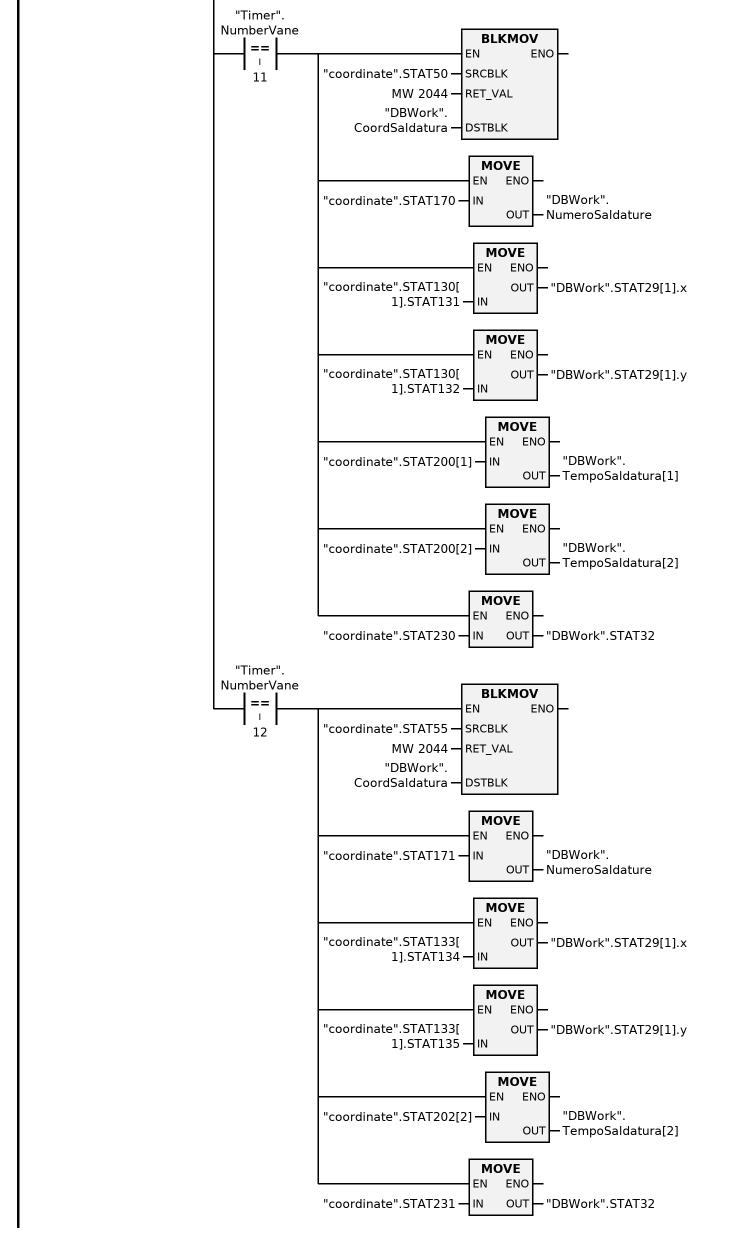
[picture p72: FC51 - TYPE TOOL networks 12-12]
NETWORK
TITLE =
      A     "Type_PP2_9_vane";
      A     "T45";
      =     L 0.0;
      A     L 0.0;
      A(;
      L     "Timer".NumberVane;
      L     9;
      ==I;
      );
      =     L 0.1;
      A     L 0.1;
      JNB   _04f;
      CALL  "BLKMOV" (
           SRCBLK                   := "coordinate".STAT40,
           RET_VAL                  := MW 2044,
           DSTBLK                   := "DBWork".CoordSaldatura);
_04f: NOP   0;
      A     L 0.1;
      JNB   _050;
      L     "coordinate".STAT168;
      T     "DBWork".NumeroSaldature;
_050: NOP   0;
      A     L 0.1;
      JNB   _051;
      L     "coordinate".STAT124[1].STAT125;
      T     "DBWork".STAT29[1].x;
_051: NOP   0;
      A     L 0.1;
      JNB   _052;
      L     "coordinate".STAT124[1].STAT126;
      T     "DBWork".STAT29[1].y;
_052: NOP   0;
      A     L 0.1;
      JNB   _053;
      L     "coordinate".STAT196[1];
      T     "DBWork".TempoSaldatura[1];
_053: NOP   0;
      A     L 0.1;
      JNB   _054;
      L     "coordinate".STAT196[2];
      T     "DBWork".TempoSaldatura[2];
_054: NOP   0;
      A     L 0.1;
      JNB   _055;
      L     "coordinate".STAT228;
      T     "DBWork".STAT32;
_055: NOP   0;
      A     L 0.0;
      A(;
      L     "Timer".NumberVane;
      L     10;
      ==I;
      );
      =     L 0.1;
      A     L 0.1;
      JNB   _056;
      CALL  "BLKMOV" (
           SRCBLK                   := "coordinate".STAT45,
           RET_VAL                  := MW 2044,
           DSTBLK                   := "DBWork".CoordSaldatura);
_056: NOP   0;
      A     L 0.1;
      JNB   _057;
      L     "coordinate".STAT169;
      T     "DBWork".NumeroSaldature;
_057: NOP   0;
      A     L 0.1;
      JNB   _058;
      L     "coordinate".STAT127[1].STAT128;
      T     "DBWork".STAT29[1].x;
_058: NOP   0;
      A     L 0.1;
      JNB   _059;
      L     "coordinate".STAT127[1].STAT129;
      T     "DBWork".STAT29[1].y;
_059: NOP   0;
      A     L 0.1;
      JNB   _05a;
      L     "coordinate".STAT198[1];
      T     "DBWork".TempoSaldatura[1];
_05a: NOP   0;
      A     L 0.1;
      JNB   _05b;
      L     "coordinate".STAT198[2];
      T     "DBWork".TempoSaldatura[2];
_05b: NOP   0;
      A     L 0.1;
      JNB   _05c;
      L     "coordinate".STAT229;
      T     "DBWork".STAT32;
_05c: NOP   0;
      A     L 0.0;
      A(;
      L     "Timer".NumberVane;
      L     11;
      ==I;
      );
      =     L 0.1;
      A     L 0.1;
      JNB   _05d;
      CALL  "BLKMOV" (
           SRCBLK                   := "coordinate".STAT50,
           RET_VAL                  := MW 2044,
           DSTBLK                   := "DBWork".CoordSaldatura);
_05d: NOP   0;
      A     L 0.1;
      JNB   _05e;
      L     "coordinate".STAT170;
      T     "DBWork".NumeroSaldature;
_05e: NOP   0;
      A     L 0.1;
      JNB   _05f;
      L     "coordinate".STAT130[1].STAT131;
      T     "DBWork".STAT29[1].x;
_05f: NOP   0;
      A     L 0.1;
      JNB   _060;
      L     "coordinate".STAT130[1].STAT132;
      T     "DBWork".STAT29[1].y;
_060: NOP   0;
      A     L 0.1;
      JNB   _061;
      L     "coordinate".STAT200[1];
      T     "DBWork".TempoSaldatura[1];
_061: NOP   0;
      A     L 0.1;
      JNB   _062;
      L     "coordinate".STAT200[2];
      T     "DBWork".TempoSaldatura[2];
_062: NOP   0;
      A     L 0.1;
      JNB   _063;
      L     "coordinate".STAT230;
      T     "DBWork".STAT32;
_063: NOP   0;
      A     L 0.0;
      A(;
      L     "Timer".NumberVane;
      L     12;
      ==I;
      );
      =     L 0.1;
      A     L 0.1;
      JNB   _064;
      CALL  "BLKMOV" (
           SRCBLK                   := "coordinate".STAT55,
           RET_VAL                  := MW 2044,
           DSTBLK                   := "DBWork".CoordSaldatura);
_064: NOP   0;
      A     L 0.1;
      JNB   _065;
      L     "coordinate".STAT171;
      T     "DBWork".NumeroSaldature;
_065: NOP   0;
      A     L 0.1;
      JNB   _066;
      L     "coordinate".STAT133[1].STAT134;
      T     "DBWork".STAT29[1].x;
_066: NOP   0;
      A     L 0.1;
      JNB   _067;
      L     "coordinate".STAT133[1].STAT135;
      T     "DBWork".STAT29[1].y;
_067: NOP   0;
      A     L 0.1;
      JNB   _068;
      L     "coordinate".STAT202[2];
      T     "DBWork".TempoSaldatura[2];
_068: NOP   0;
      A     L 0.1;
      JNB   _069;
      L     "coordinate".STAT231;
      T     "DBWork".STAT32;
_069: NOP   0;
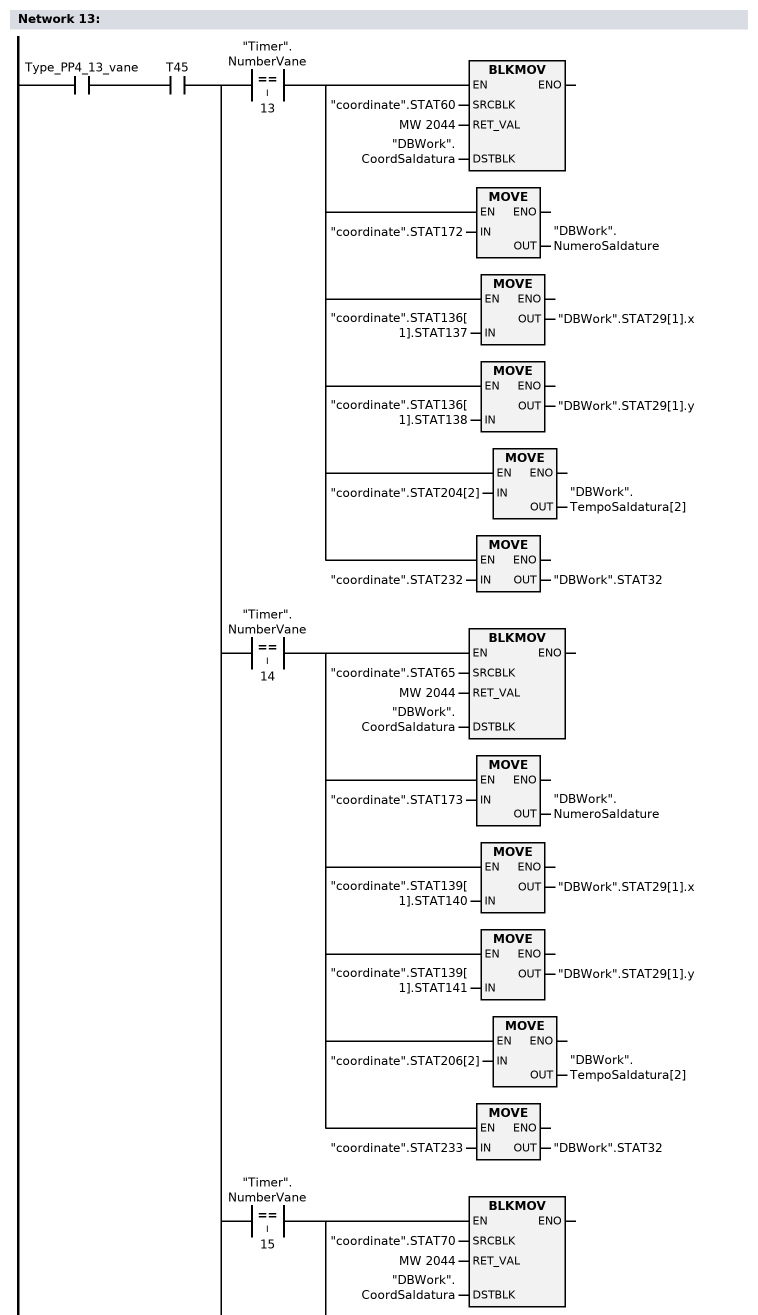
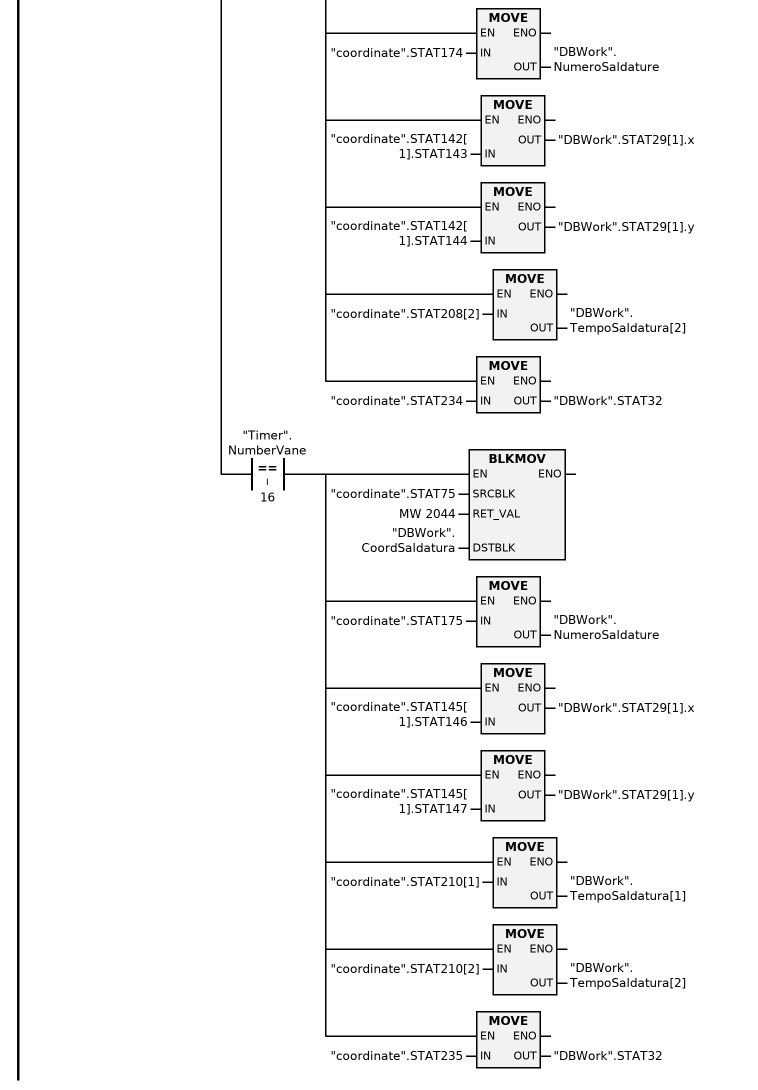
NETWORK
TITLE =
      A     "Type_PP4_13_vane";
      A     "T45";
      =     L 0.0;
      A     L 0.0;
      A(;
      L     "Timer".NumberVane;
      L     13;
      ==I;
      );
      =     L 0.1;
      A     L 0.1;
      JNB   _06a;
      CALL  "BLKMOV" (
           SRCBLK                   := "coordinate".STAT60,
           RET_VAL                  := MW 2044,
           DSTBLK                   := "DBWork".CoordSaldatura);
_06a: NOP   0;
      A     L 0.1;
      JNB   _06b;
      L     "coordinate".STAT172;
      T     "DBWork".NumeroSaldature;
_06b: NOP   0;
      A     L 0.1;
      JNB   _06c;
      L     "coordinate".STAT136[1].STAT137;
      T     "DBWork".STAT29[1].x;
_06c: NOP   0;
      A     L 0.1;
      JNB   _06d;
      L     "coordinate".STAT136[1].STAT138;
      T     "DBWork".STAT29[1].y;
_06d: NOP   0;
      A     L 0.1;
      JNB   _06e;
      L     "coordinate".STAT204[2];
      T     "DBWork".TempoSaldatura[2];
_06e: NOP   0;
      A     L 0.1;
      JNB   _06f;
      L     "coordinate".STAT232;
      T     "DBWork".STAT32;
_06f: NOP   0;
      A     L 0.0;
      A(;
      L     "Timer".NumberVane;
      L     14;
      ==I;
      );
      =     L 0.1;
      A     L 0.1;
      JNB   _070;
      CALL  "BLKMOV" (
           SRCBLK                   := "coordinate".STAT65,
           RET_VAL                  := MW 2044,
           DSTBLK                   := "DBWork".CoordSaldatura);
_070: NOP   0;
      A     L 0.1;
      JNB   _071;
      L     "coordinate".STAT173;
      T     "DBWork".NumeroSaldature;
_071: NOP   0;
      A     L 0.1;
      JNB   _072;
      L     "coordinate".STAT139[1].STAT140;
      T     "DBWork".STAT29[1].x;
_072: NOP   0;
      A     L 0.1;
      JNB   _073;
      L     "coordinate".STAT139[1].STAT141;
      T     "DBWork".STAT29[1].y;
_073: NOP   0;
      A     L 0.1;
      JNB   _074;
      L     "coordinate".STAT206[2];
      T     "DBWork".TempoSaldatura[2];
_074: NOP   0;
      A     L 0.1;
      JNB   _075;
      L     "coordinate".STAT233;
      T     "DBWork".STAT32;
_075: NOP   0;
      A     L 0.0;
      A(;
      L     "Timer".NumberVane;
      L     15;
      ==I;
      );
      =     L 0.1;
      A     L 0.1;
      JNB   _076;
      CALL  "BLKMOV" (
           SRCBLK                   := "coordinate".STAT70,
           RET_VAL                  := MW 2044,
           DSTBLK                   := "DBWork".CoordSaldatura);
_076: NOP   0;
      A     L 0.1;
      JNB   _077;
      L     "coordinate".STAT174;
      T     "DBWork".NumeroSaldature;
_077: NOP   0;
      A     L 0.1;
      JNB   _078;
      L     "coordinate".STAT142[1].STAT143;
      T     "DBWork".STAT29[1].x;
_078: NOP   0;
      A     L 0.1;
      JNB   _079;
      L     "coordinate".STAT142[1].STAT144;
      T     "DBWork".STAT29[1].y;
_079: NOP   0;
      A     L 0.1;
      JNB   _07a;
      L     "coordinate".STAT208[2];
      T     "DBWork".TempoSaldatura[2];
_07a: NOP   0;
      A     L 0.1;
      JNB   _07b;
      L     "coordinate".STAT234;
      T     "DBWork".STAT32;
_07b: NOP   0;
      A     L 0.0;
      A(;
      L     "Timer".NumberVane;
      L     16;
      ==I;
      );
      =     L 0.1;
      A     L 0.1;
      JNB   _07c;
      CALL  "BLKMOV" (
           SRCBLK                   := "coordinate".STAT75,
           RET_VAL                  := MW 2044,
           DSTBLK                   := "DBWork".CoordSaldatura);
_07c: NOP   0;
      A     L 0.1;
      JNB   _07d;
      L     "coordinate".STAT175;
      T     "DBWork".NumeroSaldature;
_07d: NOP   0;
      A     L 0.1;
      JNB   _07e;
      L     "coordinate".STAT145[1].STAT146;
      T     "DBWork".STAT29[1].x;
_07e: NOP   0;
      A     L 0.1;
      JNB   _07f;
      L     "coordinate".STAT145[1].STAT147;
      T     "DBWork".STAT29[1].y;
_07f: NOP   0;
      A     L 0.1;
      JNB   _080;
      L     "coordinate".STAT210[1];
      T     "DBWork".TempoSaldatura[1];
_080: NOP   0;
      A     L 0.1;
      JNB   _081;
      L     "coordinate".STAT210[2];
      T     "DBWork".TempoSaldatura[2];
_081: NOP   0;
      A     L 0.1;
      JNB   _082;
      L     "coordinate".STAT235;
      T     "DBWork".STAT32;
_082: NOP   0;
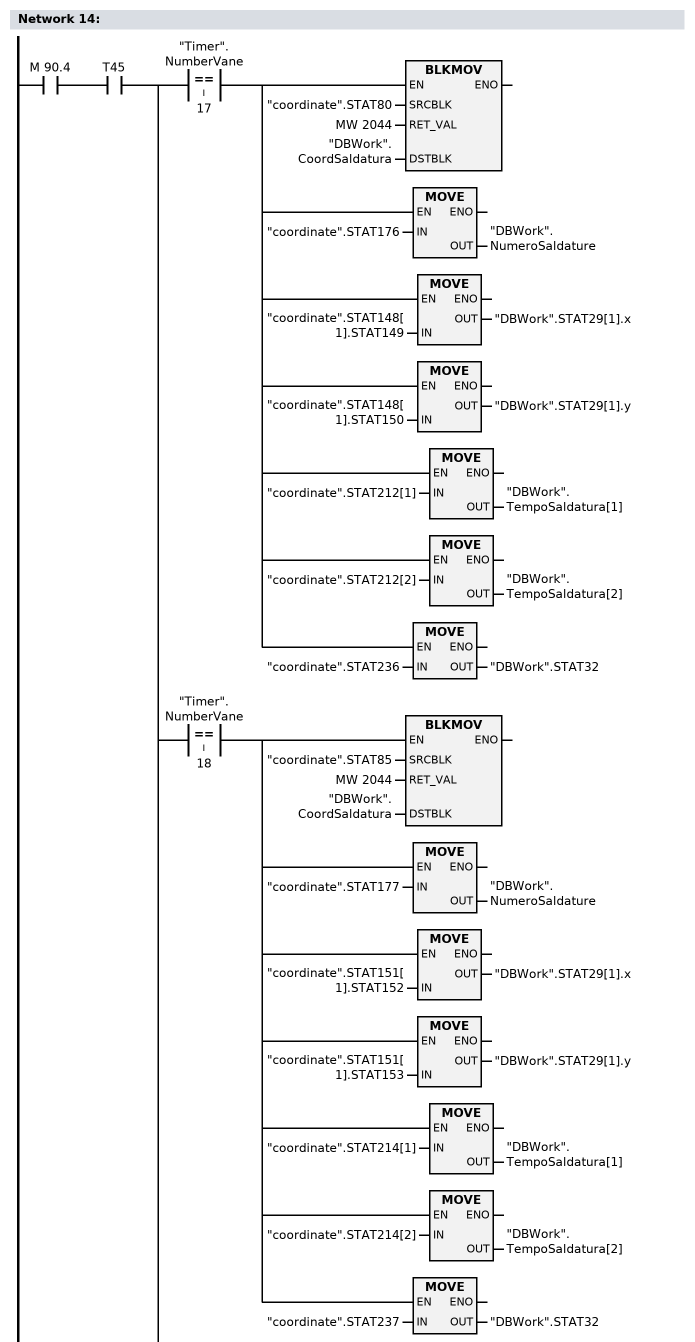
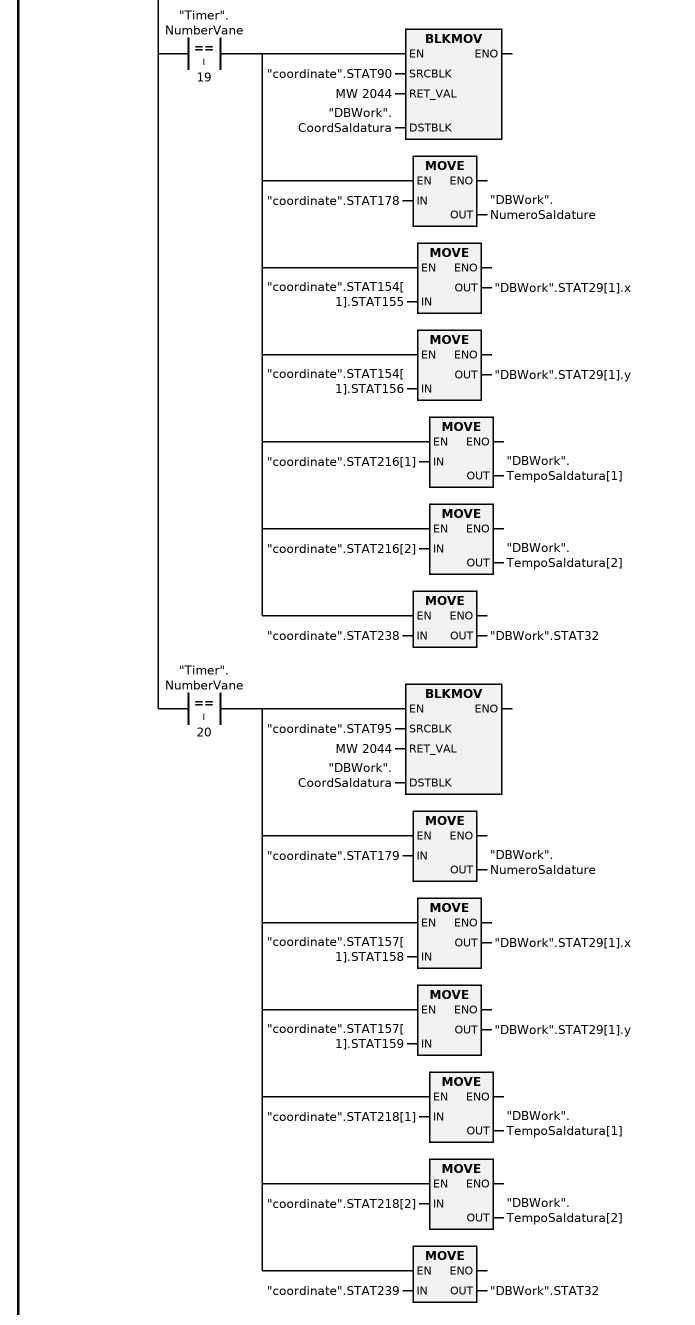
NETWORK
TITLE =
      A     M 90.4;
      A     "T45";
      =     L 0.0;
      A     L 0.0;
      A(;
      L     "Timer".NumberVane;
      L     17;
      ==I;
      );
      =     L 0.1;
      A     L 0.1;
      JNB   _083;
      CALL  "BLKMOV" (
           SRCBLK                   := "coordinate".STAT80,
           RET_VAL                  := MW 2044,
           DSTBLK                   := "DBWork".CoordSaldatura);
_083: NOP   0;
      A     L 0.1;
      JNB   _084;
      L     "coordinate".STAT176;
      T     "DBWork".NumeroSaldature;
_084: NOP   0;
      A     L 0.1;
      JNB   _085;
      L     "coordinate".STAT148[1].STAT149;
      T     "DBWork".STAT29[1].x;
_085: NOP   0;
      A     L 0.1;
      JNB   _086;
      L     "coordinate".STAT148[1].STAT150;
      T     "DBWork".STAT29[1].y;
_086: NOP   0;
      A     L 0.1;
      JNB   _087;
      L     "coordinate".STAT212[1];
      T     "DBWork".TempoSaldatura[1];
_087: NOP   0;
      A     L 0.1;
      JNB   _088;
      L     "coordinate".STAT212[2];
      T     "DBWork".TempoSaldatura[2];
_088: NOP   0;
      A     L 0.1;
      JNB   _089;
      L     "coordinate".STAT236;
      T     "DBWork".STAT32;
_089: NOP   0;
      A     L 0.0;
      A(;
      L     "Timer".NumberVane;
      L     18;
      ==I;
      );
      =     L 0.1;
      A     L 0.1;
      JNB   _08a;
      CALL  "BLKMOV" (
           SRCBLK                   := "coordinate".STAT85,
           RET_VAL                  := MW 2044,
           DSTBLK                   := "DBWork".CoordSaldatura);
_08a: NOP   0;
      A     L 0.1;
      JNB   _08b;
      L     "coordinate".STAT177;
      T     "DBWork".NumeroSaldature;
_08b: NOP   0;
      A     L 0.1;
      JNB   _08c;
      L     "coordinate".STAT151[1].STAT152;
      T     "DBWork".STAT29[1].x;
_08c: NOP   0;
      A     L 0.1;
      JNB   _08d;
      L     "coordinate".STAT151[1].STAT153;
      T     "DBWork".STAT29[1].y;
_08d: NOP   0;
      A     L 0.1;
      JNB   _08e;
      L     "coordinate".STAT214[1];
      T     "DBWork".TempoSaldatura[1];
_08e: NOP   0;
      A     L 0.1;
      JNB   _08f;
      L     "coordinate".STAT214[2];
      T     "DBWork".TempoSaldatura[2];
_08f: NOP   0;
      A     L 0.1;
      JNB   _090;
      L     "coordinate".STAT237;
      T     "DBWork".STAT32;
_090: NOP   0;
      A     L 0.0;
      A(;
      L     "Timer".NumberVane;
      L     19;
      ==I;
      );
      =     L 0.1;
      A     L 0.1;
      JNB   _091;
      CALL  "BLKMOV" (
           SRCBLK                   := "coordinate".STAT90,
           RET_VAL                  := MW 2044,
           DSTBLK                   := "DBWork".CoordSaldatura);
_091: NOP   0;
      A     L 0.1;
      JNB   _092;
      L     "coordinate".STAT178;
      T     "DBWork".NumeroSaldature;
_092: NOP   0;
      A     L 0.1;
      JNB   _093;
      L     "coordinate".STAT154[1].STAT155;
      T     "DBWork".STAT29[1].x;
_093: NOP   0;
      A     L 0.1;
      JNB   _094;
      L     "coordinate".STAT154[1].STAT156;
      T     "DBWork".STAT29[1].y;
_094: NOP   0;
      A     L 0.1;
      JNB   _095;
      L     "coordinate".STAT216[1];
      T     "DBWork".TempoSaldatura[1];
_095: NOP   0;
      A     L 0.1;
      JNB   _096;
      L     "coordinate".STAT216[2];
      T     "DBWork".TempoSaldatura[2];
_096: NOP   0;
      A     L 0.1;
      JNB   _097;
      L     "coordinate".STAT238;
      T     "DBWork".STAT32;
_097: NOP   0;
      A     L 0.0;
      A(;
      L     "Timer".NumberVane;
      L     20;
      ==I;
      );
      =     L 0.1;
      A     L 0.1;
      JNB   _098;
      CALL  "BLKMOV" (
           SRCBLK                   := "coordinate".STAT95,
           RET_VAL                  := MW 2044,
           DSTBLK                   := "DBWork".CoordSaldatura);
_098: NOP   0;
      A     L 0.1;
      JNB   _099;
      L     "coordinate".STAT179;
      T     "DBWork".NumeroSaldature;
_099: NOP   0;
      A     L 0.1;
      JNB   _09a;
      L     "coordinate".STAT157[1].STAT158;
      T     "DBWork".STAT29[1].x;
_09a: NOP   0;
      A     L 0.1;
      JNB   _09b;
      L     "coordinate".STAT157[1].STAT159;
      T     "DBWork".STAT29[1].y;
_09b: NOP   0;
      A     L 0.1;
      JNB   _09c;
      L     "coordinate".STAT218[1];
      T     "DBWork".TempoSaldatura[1];
_09c: NOP   0;
      A     L 0.1;
      JNB   _09d;
      L     "coordinate".STAT218[2];
      T     "DBWork".TempoSaldatura[2];
_09d: NOP   0;
      A     L 0.1;
      JNB   _09e;
      L     "coordinate".STAT239;
      T     "DBWork".STAT32;
_09e: NOP   0;
END_FUNCTION

FUNCTION "FC52 - SYSTEM VISION" : VOID	// FC 52
VERSION : 0.1
BEGIN
// (block stored without names or comments; labels and parameter names are numbered)
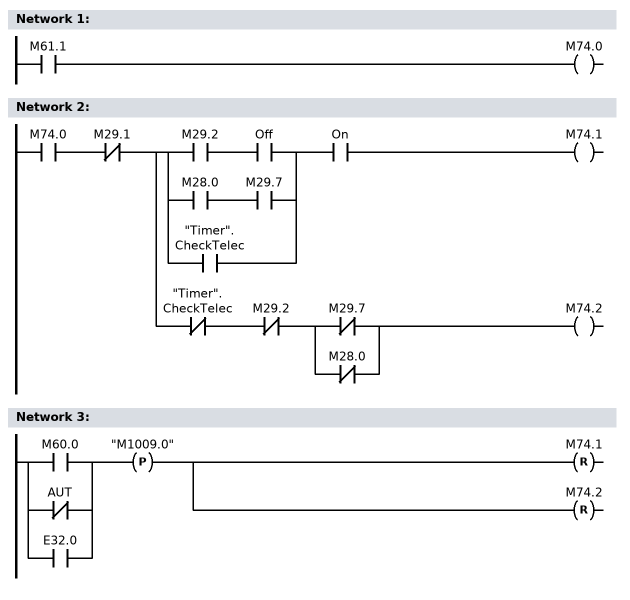
NETWORK
TITLE =
      A     "M61.1";
      =     "M74.0";
NETWORK
TITLE =
      A     "M74.0";
      AN    "M29.1";
      =     L 0.0;
      A     L 0.0;
      A(;
      A     "M29.2";
      A     "Off";
      O;
      A     "M28.0";
      A     "M29.7";
      O     "Timer".CheckTelec;
      );
      A     "On";
      =     "M74.1";
      A     L 0.0;
      AN    "Timer".CheckTelec;
      AN    "M29.2";
      A(;
      ON    "M29.7";
      ON    "M28.0";
      );
      =     "M74.2";
NETWORK
TITLE =
      A(;
      O     "M60.0";
      ON    "AUT";
      O     "E32.0";
      );
      FP    "M1009.0";
      R     "M74.1";
      R     "M74.2";
END_FUNCTION

FUNCTION "FC53 - REWORK" : VOID	// FC 53
VERSION : 0.1
BEGIN
NETWORK
TITLE =
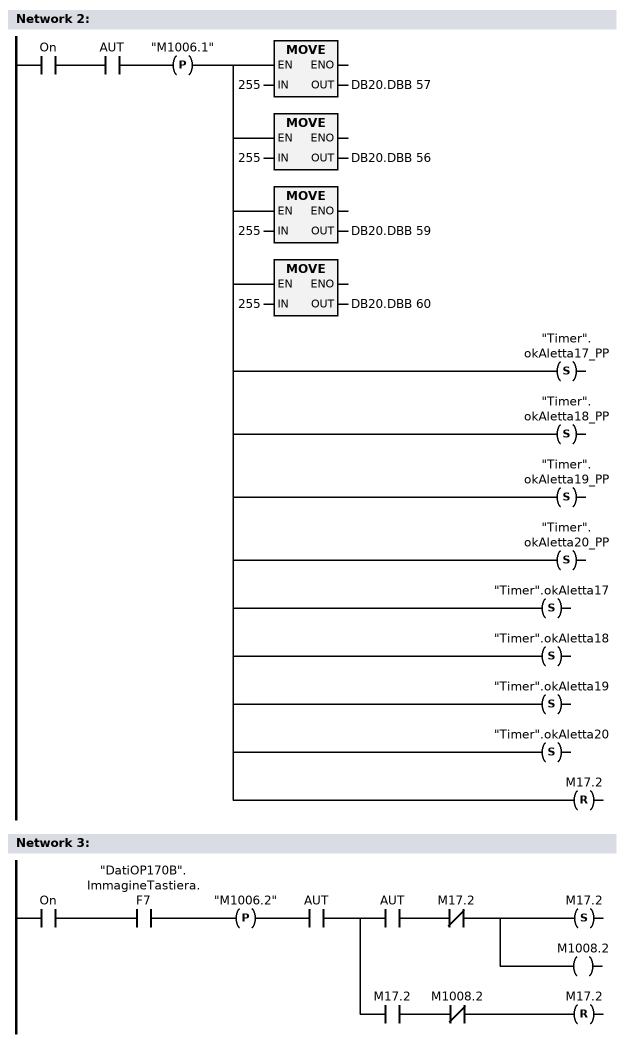
NETWORK
TITLE =
      A     "On";
      A     "AUT";
      FP    "M1006.1";
      =     L 0.0;
      A     L 0.0;
      JNB   _001;
      L     255;
      T     DB20.DBB 57;
_001: NOP   0;
      A     L 0.0;
      JNB   _002;
      L     255;
      T     DB20.DBB 56;
_002: NOP   0;
      A     L 0.0;
      JNB   _003;
      L     255;
      T     DB20.DBB 59;
_003: NOP   0;
      A     L 0.0;
      JNB   _004;
      L     255;
      T     DB20.DBB 60;
_004: NOP   0;
      A     L 0.0;
      BLD   102;
      S     "Timer".okAletta17_PP;
      A     L 0.0;
      BLD   102;
      S     "Timer".okAletta18_PP;
      A     L 0.0;
      BLD   102;
      S     "Timer".okAletta19_PP;
      A     L 0.0;
      BLD   102;
      S     "Timer".okAletta20_PP;
      A     L 0.0;
      BLD   102;
      S     "Timer".okAletta17;
      A     L 0.0;
      BLD   102;
      S     "Timer".okAletta18;
      A     L 0.0;
      BLD   102;
      S     "Timer".okAletta19;
      A     L 0.0;
      BLD   102;
      S     "Timer".okAletta20;
      A     L 0.0;
      BLD   102;
      R     "M17.2";
NETWORK
TITLE =
      A     "On";
      A     "DatiOP170B".ImmagineTastiera.F7;
      FP    "M1006.2";
      A     "AUT";
      =     L 0.0;
      A     L 0.0;
      A     "AUT";
      AN    "M17.2";
      S     "M17.2";
      =     "M1008.2";
      A     L 0.0;
      A     "M17.2";
      AN    "M1008.2";
      R     "M17.2";
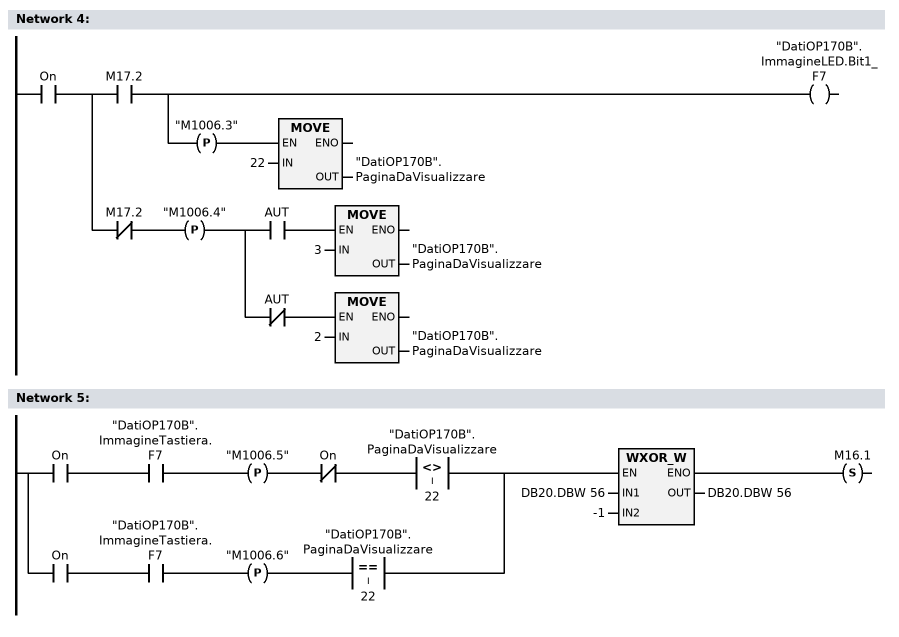
NETWORK
TITLE =
      A     "On";
      =     L 0.0;
      A     L 0.0;
      A     "M17.2";
      =     L 0.1;
      A     L 0.1;
      BLD   102;
      =     "DatiOP170B".ImmagineLED.Bit1_F7;
      A     L 0.1;
      FP    "M1006.3";
      JNB   _005;
      L     22;
      T     "DatiOP170B".PaginaDaVisualizzare;
_005: NOP   0;
      A     L 0.0;
      AN    "M17.2";
      FP    "M1006.4";
      =     L 0.1;
      A     L 0.1;
      A     "AUT";
      JNB   _006;
      L     3;
      T     "DatiOP170B".PaginaDaVisualizzare;
_006: NOP   0;
      A     L 0.1;
      AN    "AUT";
      JNB   _007;
      L     2;
      T     "DatiOP170B".PaginaDaVisualizzare;
_007: NOP   0;
NETWORK
TITLE =
      A(;
      A     "On";
      A     "DatiOP170B".ImmagineTastiera.F7;
      FP    "M1006.5";
      AN    "On";
      A(;
      L     "DatiOP170B".PaginaDaVisualizzare;
      L     22;
      <>I;
      );
      O(;
      A     "On";
      A     "DatiOP170B".ImmagineTastiera.F7;
      FP    "M1006.6";
      A(;
      L     "DatiOP170B".PaginaDaVisualizzare;
      L     22;
      ==I;
      );
      );
      );
      JNB   _008;
      L     DB20.DBW 56;
      L     -1;
      XOW;
      T     DB20.DBW 56;
      SET;
      SAVE;
      CLR;
_008: A     BR;
      S     "M16.1";
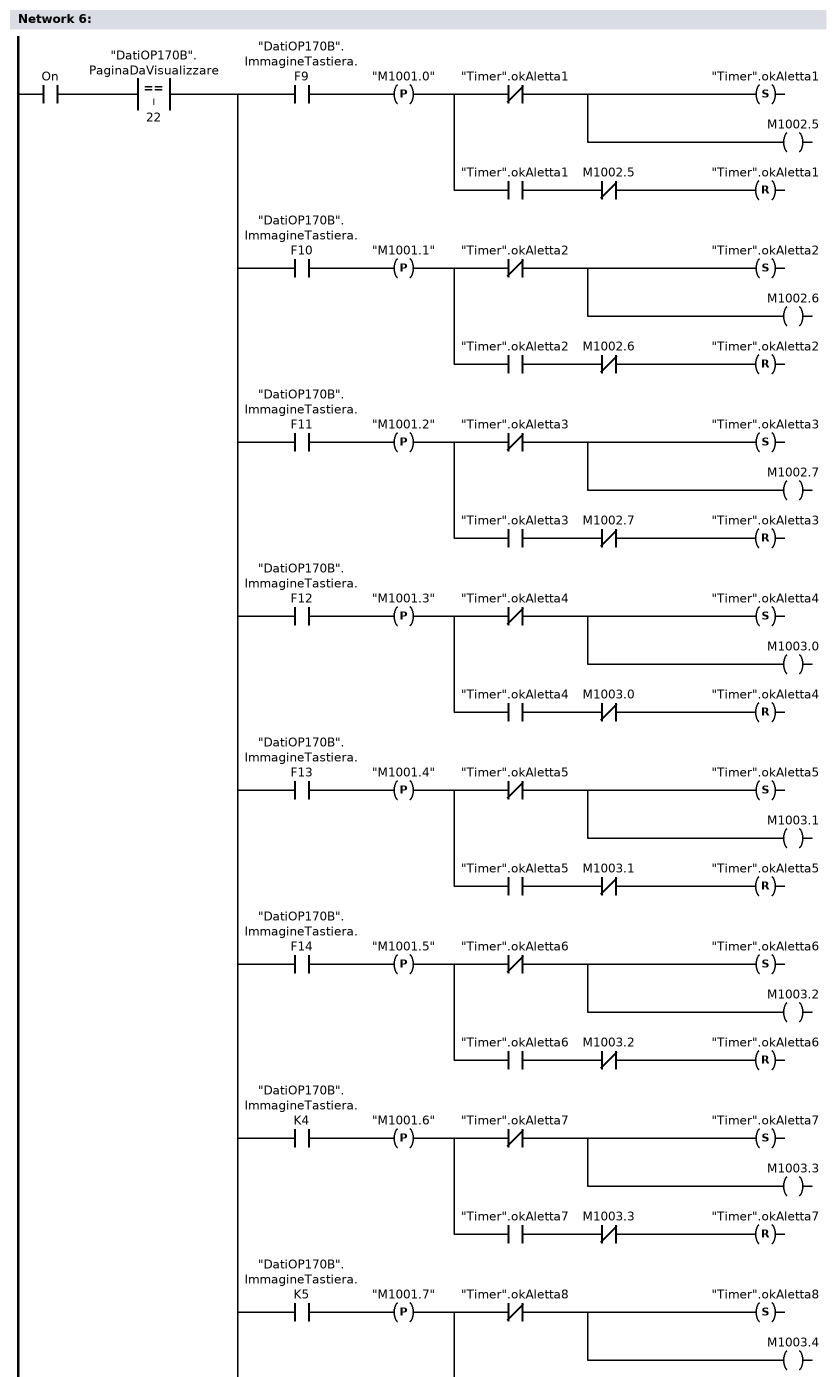
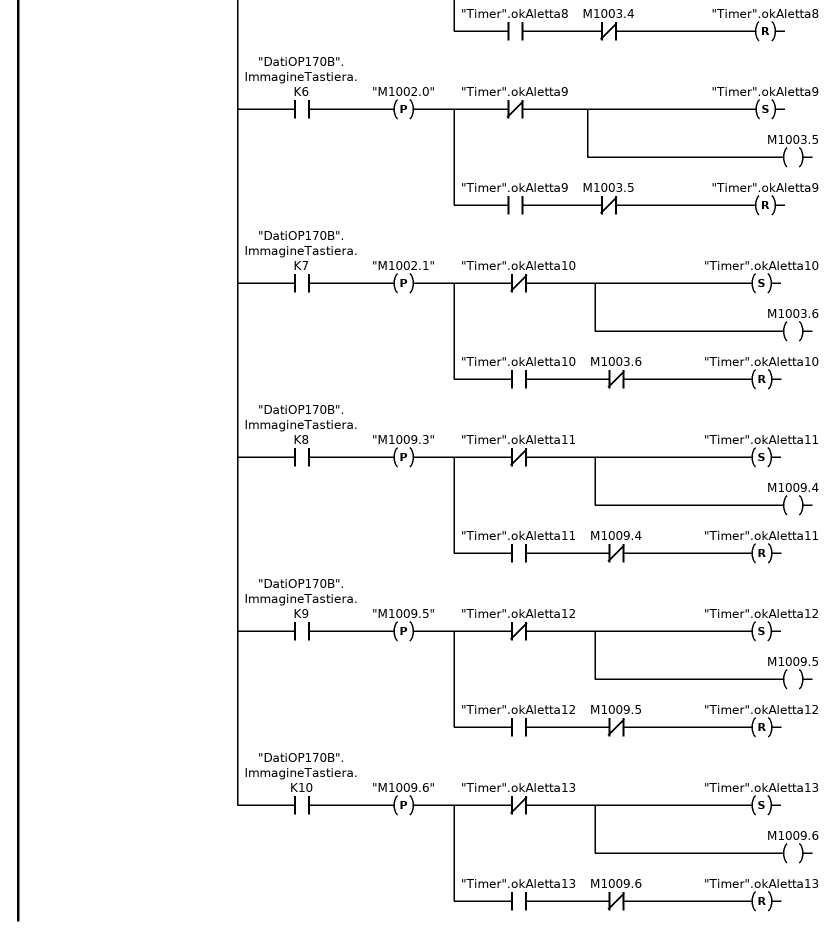
NETWORK
TITLE =
      A     "On";
      A(;
      L     "DatiOP170B".PaginaDaVisualizzare;
      L     22;
      ==I;
      );
      =     L 0.0;
      A     L 0.0;
      A     "DatiOP170B".ImmagineTastiera.F9;
      FP    "M1001.0";
      =     L 0.1;
      A     L 0.1;
      AN    "Timer".okAletta1;
      S     "Timer".okAletta1;
      =     "M1002.5";
      A     L 0.1;
      A     "Timer".okAletta1;
      AN    "M1002.5";
      R     "Timer".okAletta1;
      A     L 0.0;
      A     "DatiOP170B".ImmagineTastiera.F10;
      FP    "M1001.1";
      =     L 0.1;
      A     L 0.1;
      AN    "Timer".okAletta2;
      S     "Timer".okAletta2;
      =     "M1002.6";
      A     L 0.1;
      A     "Timer".okAletta2;
      AN    "M1002.6";
      R     "Timer".okAletta2;
      A     L 0.0;
      A     "DatiOP170B".ImmagineTastiera.F11;
      FP    "M1001.2";
      =     L 0.1;
      A     L 0.1;
      AN    "Timer".okAletta3;
      S     "Timer".okAletta3;
      =     "M1002.7";
      A     L 0.1;
      A     "Timer".okAletta3;
      AN    "M1002.7";
      R     "Timer".okAletta3;
      A     L 0.0;
      A     "DatiOP170B".ImmagineTastiera.F12;
      FP    "M1001.3";
      =     L 0.1;
      A     L 0.1;
      AN    "Timer".okAletta4;
      S     "Timer".okAletta4;
      =     "M1003.0";
      A     L 0.1;
      A     "Timer".okAletta4;
      AN    "M1003.0";
      R     "Timer".okAletta4;
      A     L 0.0;
      A     "DatiOP170B".ImmagineTastiera.F13;
      FP    "M1001.4";
      =     L 0.1;
      A     L 0.1;
      AN    "Timer".okAletta5;
      S     "Timer".okAletta5;
      =     "M1003.1";
      A     L 0.1;
      A     "Timer".okAletta5;
      AN    "M1003.1";
      R     "Timer".okAletta5;
      A     L 0.0;
      A     "DatiOP170B".ImmagineTastiera.F14;
      FP    "M1001.5";
      =     L 0.1;
      A     L 0.1;
      AN    "Timer".okAletta6;
      S     "Timer".okAletta6;
      =     "M1003.2";
      A     L 0.1;
      A     "Timer".okAletta6;
      AN    "M1003.2";
      R     "Timer".okAletta6;
      A     L 0.0;
      A     "DatiOP170B".ImmagineTastiera.K4;
      FP    "M1001.6";
      =     L 0.1;
      A     L 0.1;
      AN    "Timer".okAletta7;
      S     "Timer".okAletta7;
      =     "M1003.3";
      A     L 0.1;
      A     "Timer".okAletta7;
      AN    "M1003.3";
      R     "Timer".okAletta7;
      A     L 0.0;
      A     "DatiOP170B".ImmagineTastiera.K5;
      FP    "M1001.7";
      =     L 0.1;
      A     L 0.1;
      AN    "Timer".okAletta8;
      S     "Timer".okAletta8;
      =     "M1003.4";
      A     L 0.1;
      A     "Timer".okAletta8;
      AN    "M1003.4";
      R     "Timer".okAletta8;
      A     L 0.0;
      A     "DatiOP170B".ImmagineTastiera.K6;
      FP    "M1002.0";
      =     L 0.1;
      A     L 0.1;
      AN    "Timer".okAletta9;
      S     "Timer".okAletta9;
      =     "M1003.5";
      A     L 0.1;
      A     "Timer".okAletta9;
      AN    "M1003.5";
      R     "Timer".okAletta9;
      A     L 0.0;
      A     "DatiOP170B".ImmagineTastiera.K7;
      FP    "M1002.1";
      =     L 0.1;
      A     L 0.1;
      AN    "Timer".okAletta10;
      S     "Timer".okAletta10;
      =     "M1003.6";
      A     L 0.1;
      A     "Timer".okAletta10;
      AN    "M1003.6";
      R     "Timer".okAletta10;
      A     L 0.0;
      A     "DatiOP170B".ImmagineTastiera.K8;
      FP    "M1009.3";
      =     L 0.1;
      A     L 0.1;
      AN    "Timer".okAletta11;
      S     "Timer".okAletta11;
      =     "M1009.4";
      A     L 0.1;
      A     "Timer".okAletta11;
      AN    "M1009.4";
      R     "Timer".okAletta11;
      A     L 0.0;
      A     "DatiOP170B".ImmagineTastiera.K9;
      FP    "M1009.5";
      =     L 0.1;
      A     L 0.1;
      AN    "Timer".okAletta12;
      S     "Timer".okAletta12;
      =     "M1009.5";
      A     L 0.1;
      A     "Timer".okAletta12;
      AN    "M1009.5";
      R     "Timer".okAletta12;
      A     L 0.0;
      A     "DatiOP170B".ImmagineTastiera.K10;
      FP    "M1009.6";
      =     L 0.1;
      A     L 0.1;
      AN    "Timer".okAletta13;
      S     "Timer".okAletta13;
      =     "M1009.6";
      A     L 0.1;
      A     "Timer".okAletta13;
      AN    "M1009.6";
      R     "Timer".okAletta13;
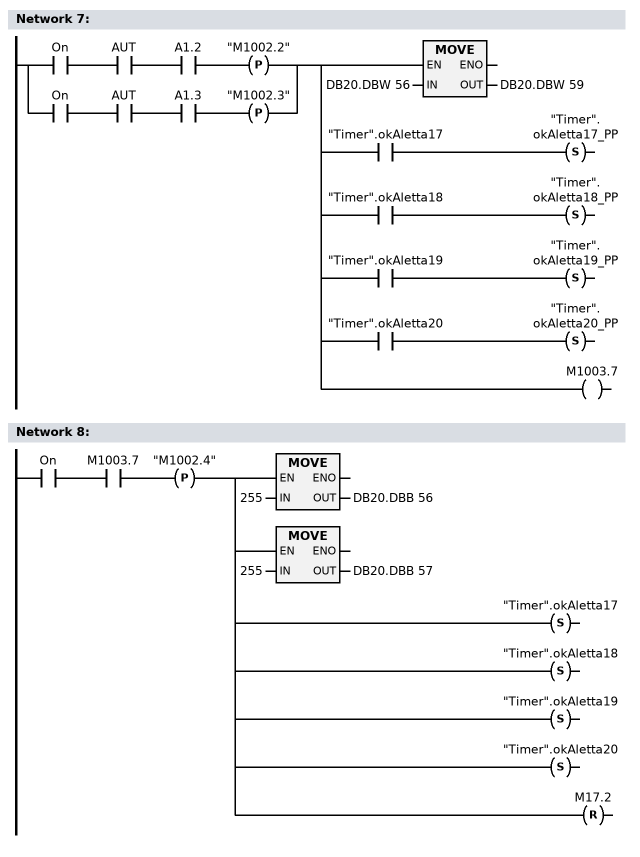
NETWORK
TITLE =
      A     "On";
      A     "AUT";
      A     "A1.2";
      FP    "M1002.2";
      O(;
      A     "On";
      A     "AUT";
      A     "A1.3";
      FP    "M1002.3";
      );
      =     L 0.0;
      A     L 0.0;
      JNB   _009;
      L     DB20.DBW 56;
      T     DB20.DBW 59;
_009: NOP   0;
      A     L 0.0;
      A     "Timer".okAletta17;
      S     "Timer".okAletta17_PP;
      A     L 0.0;
      A     "Timer".okAletta18;
      S     "Timer".okAletta18_PP;
      A     L 0.0;
      A     "Timer".okAletta19;
      S     "Timer".okAletta19_PP;
      A     L 0.0;
      A     "Timer".okAletta20;
      S     "Timer".okAletta20_PP;
      A     L 0.0;
      BLD   102;
      =     "M1003.7";
NETWORK
TITLE =
      A     "On";
      A     "M1003.7";
      FP    "M1002.4";
      =     L 0.0;
      A     L 0.0;
      JNB   _00a;
      L     255;
      T     DB20.DBB 56;
_00a: NOP   0;
      A     L 0.0;
      JNB   _00b;
      L     255;
      T     DB20.DBB 57;
_00b: NOP   0;
      A     L 0.0;
      BLD   102;
      S     "Timer".okAletta17;
      A     L 0.0;
      BLD   102;
      S     "Timer".okAletta18;
      A     L 0.0;
      BLD   102;
      S     "Timer".okAletta19;
      A     L 0.0;
      BLD   102;
      S     "Timer".okAletta20;
      A     L 0.0;
      BLD   102;
      R     "M17.2";
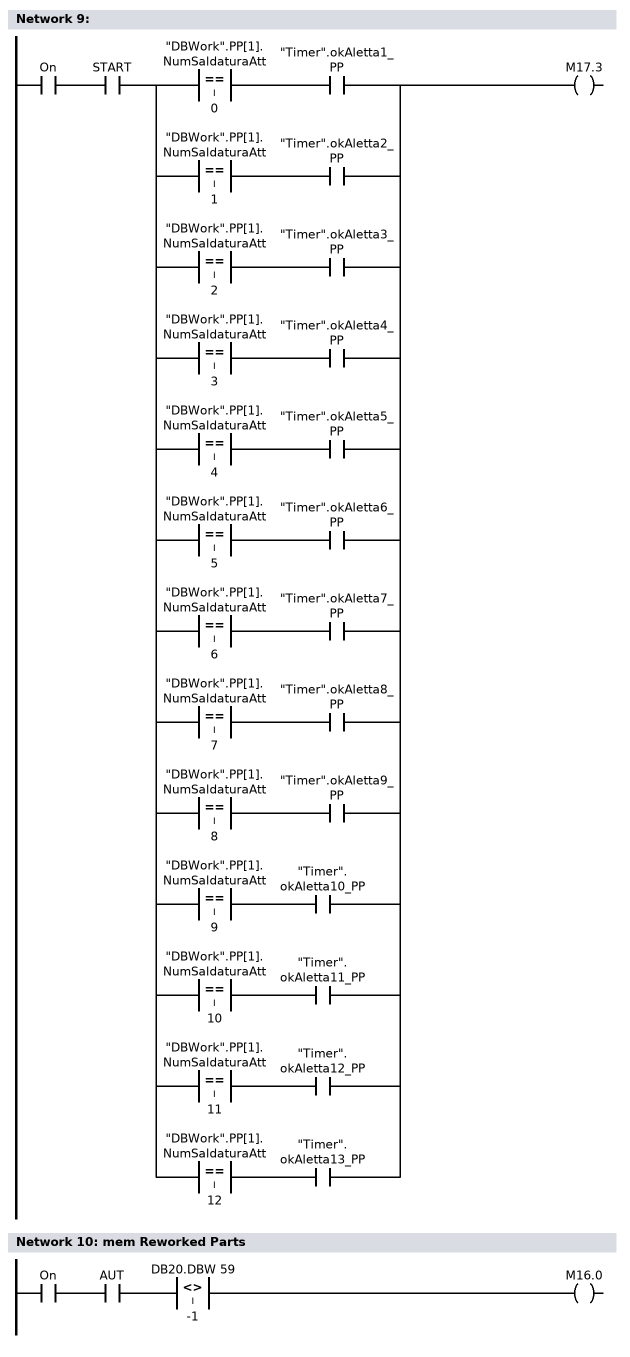
NETWORK
TITLE =
      A     "On";
      A     "START";
      A(;
      A(;
      L     "DBWork".PP[1].NumSaldaturaAtt;
      L     0;
      ==I;
      );
      A     "Timer".okAletta1_PP;
      O;
      A(;
      L     "DBWork".PP[1].NumSaldaturaAtt;
      L     1;
      ==I;
      );
      A     "Timer".okAletta2_PP;
      O;
      A(;
      L     "DBWork".PP[1].NumSaldaturaAtt;
      L     2;
      ==I;
      );
      A     "Timer".okAletta3_PP;
      O;
      A(;
      L     "DBWork".PP[1].NumSaldaturaAtt;
      L     3;
      ==I;
      );
      A     "Timer".okAletta4_PP;
      O;
      A(;
      L     "DBWork".PP[1].NumSaldaturaAtt;
      L     4;
      ==I;
      );
      A     "Timer".okAletta5_PP;
      O;
      A(;
      L     "DBWork".PP[1].NumSaldaturaAtt;
      L     5;
      ==I;
      );
      A     "Timer".okAletta6_PP;
      O;
      A(;
      L     "DBWork".PP[1].NumSaldaturaAtt;
      L     6;
      ==I;
      );
      A     "Timer".okAletta7_PP;
      O;
      A(;
      L     "DBWork".PP[1].NumSaldaturaAtt;
      L     7;
      ==I;
      );
      A     "Timer".okAletta8_PP;
      O;
      A(;
      L     "DBWork".PP[1].NumSaldaturaAtt;
      L     8;
      ==I;
      );
      A     "Timer".okAletta9_PP;
      O;
      A(;
      L     "DBWork".PP[1].NumSaldaturaAtt;
      L     9;
      ==I;
      );
      A     "Timer".okAletta10_PP;
      O;
      A(;
      L     "DBWork".PP[1].NumSaldaturaAtt;
      L     10;
      ==I;
      );
      A     "Timer".okAletta11_PP;
      O;
      A(;
      L     "DBWork".PP[1].NumSaldaturaAtt;
      L     11;
      ==I;
      );
      A     "Timer".okAletta12_PP;
      O;
      A(;
      L     "DBWork".PP[1].NumSaldaturaAtt;
      L     12;
      ==I;
      );
      A     "Timer".okAletta13_PP;
      );
      =     "M17.3";
NETWORK
TITLE = mem Reworked Parts
      A     "On";
      A     "AUT";
      A(;
      L     DB20.DBW 59;
      L     -1;
      <>I;
      );
      =     "M16.0";
END_FUNCTION

FUNCTION FC 54 : VOID
VERSION : 0.1
BEGIN
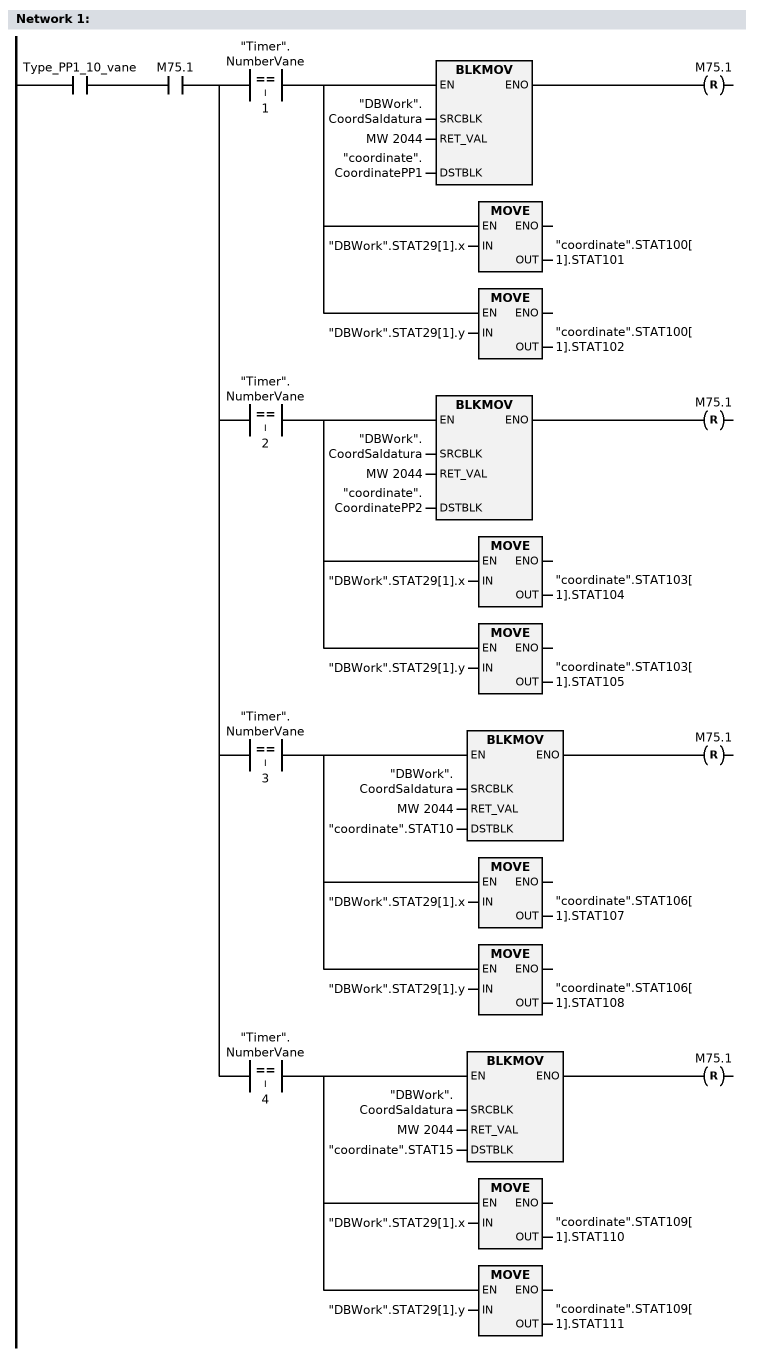
NETWORK
TITLE =
      A     "Type_PP1_10_vane";
      A     "M75.1";
      =     L 0.0;
      A     L 0.0;
      A(;
      L     "Timer".NumberVane;
      L     1;
      ==I;
      );
      =     L 0.1;
      A     L 0.1;
      JNB   _001;
      CALL  "BLKMOV" (
           SRCBLK                   := "DBWork".CoordSaldatura,
           RET_VAL                  := MW 2044,
           DSTBLK                   := "coordinate".CoordinatePP1);
_001: A     BR;
      R     "M75.1";
      A     L 0.1;
      JNB   _002;
      L     "DBWork".STAT29[1].x;
      T     "coordinate".STAT100[1].STAT101;
_002: NOP   0;
      A     L 0.1;
      JNB   _003;
      L     "DBWork".STAT29[1].y;
      T     "coordinate".STAT100[1].STAT102;
_003: NOP   0;
      A     L 0.0;
      A(;
      L     "Timer".NumberVane;
      L     2;
      ==I;
      );
      =     L 0.1;
      A     L 0.1;
      JNB   _004;
      CALL  "BLKMOV" (
           SRCBLK                   := "DBWork".CoordSaldatura,
           RET_VAL                  := MW 2044,
           DSTBLK                   := "coordinate".CoordinatePP2);
_004: A     BR;
      R     "M75.1";
      A     L 0.1;
      JNB   _005;
      L     "DBWork".STAT29[1].x;
      T     "coordinate".STAT103[1].STAT104;
_005: NOP   0;
      A     L 0.1;
      JNB   _006;
      L     "DBWork".STAT29[1].y;
      T     "coordinate".STAT103[1].STAT105;
_006: NOP   0;
      A     L 0.0;
      A(;
      L     "Timer".NumberVane;
      L     3;
      ==I;
      );
      =     L 0.1;
      A     L 0.1;
      JNB   _007;
      CALL  "BLKMOV" (
           SRCBLK                   := "DBWork".CoordSaldatura,
           RET_VAL                  := MW 2044,
           DSTBLK                   := "coordinate".STAT10);
_007: A     BR;
      R     "M75.1";
      A     L 0.1;
      JNB   _008;
      L     "DBWork".STAT29[1].x;
      T     "coordinate".STAT106[1].STAT107;
_008: NOP   0;
      A     L 0.1;
      JNB   _009;
      L     "DBWork".STAT29[1].y;
      T     "coordinate".STAT106[1].STAT108;
_009: NOP   0;
      A     L 0.0;
      A(;
      L     "Timer".NumberVane;
      L     4;
      ==I;
      );
      =     L 0.1;
      A     L 0.1;
      JNB   _00a;
      CALL  "BLKMOV" (
           SRCBLK                   := "DBWork".CoordSaldatura,
           RET_VAL                  := MW 2044,
           DSTBLK                   := "coordinate".STAT15);
_00a: A     BR;
      R     "M75.1";
      A     L 0.1;
      JNB   _00b;
      L     "DBWork".STAT29[1].x;
      T     "coordinate".STAT109[1].STAT110;
_00b: NOP   0;
      A     L 0.1;
      JNB   _00c;
      L     "DBWork".STAT29[1].y;
      T     "coordinate".STAT109[1].STAT111;
_00c: NOP   0;
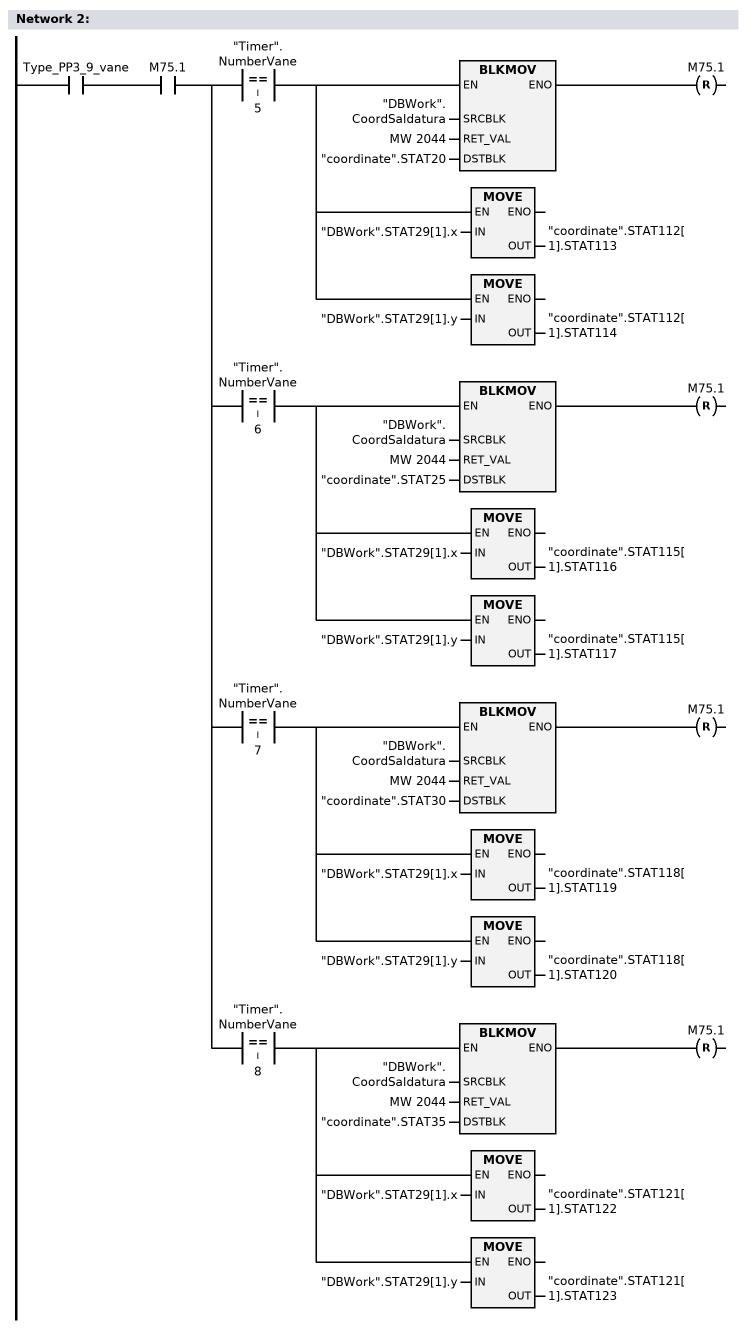
NETWORK
TITLE =
      A     "Type_PP3_9_vane";
      A     "M75.1";
      =     L 0.0;
      A     L 0.0;
      A(;
      L     "Timer".NumberVane;
      L     5;
      ==I;
      );
      =     L 0.1;
      A     L 0.1;
      JNB   _00d;
      CALL  "BLKMOV" (
           SRCBLK                   := "DBWork".CoordSaldatura,
           RET_VAL                  := MW 2044,
           DSTBLK                   := "coordinate".STAT20);
_00d: A     BR;
      R     "M75.1";
      A     L 0.1;
      JNB   _00e;
      L     "DBWork".STAT29[1].x;
      T     "coordinate".STAT112[1].STAT113;
_00e: NOP   0;
      A     L 0.1;
      JNB   _00f;
      L     "DBWork".STAT29[1].y;
      T     "coordinate".STAT112[1].STAT114;
_00f: NOP   0;
      A     L 0.0;
      A(;
      L     "Timer".NumberVane;
      L     6;
      ==I;
      );
      =     L 0.1;
      A     L 0.1;
      JNB   _010;
      CALL  "BLKMOV" (
           SRCBLK                   := "DBWork".CoordSaldatura,
           RET_VAL                  := MW 2044,
           DSTBLK                   := "coordinate".STAT25);
_010: A     BR;
      R     "M75.1";
      A     L 0.1;
      JNB   _011;
      L     "DBWork".STAT29[1].x;
      T     "coordinate".STAT115[1].STAT116;
_011: NOP   0;
      A     L 0.1;
      JNB   _012;
      L     "DBWork".STAT29[1].y;
      T     "coordinate".STAT115[1].STAT117;
_012: NOP   0;
      A     L 0.0;
      A(;
      L     "Timer".NumberVane;
      L     7;
      ==I;
      );
      =     L 0.1;
      A     L 0.1;
      JNB   _013;
      CALL  "BLKMOV" (
           SRCBLK                   := "DBWork".CoordSaldatura,
           RET_VAL                  := MW 2044,
           DSTBLK                   := "coordinate".STAT30);
_013: A     BR;
      R     "M75.1";
      A     L 0.1;
      JNB   _014;
      L     "DBWork".STAT29[1].x;
      T     "coordinate".STAT118[1].STAT119;
_014: NOP   0;
      A     L 0.1;
      JNB   _015;
      L     "DBWork".STAT29[1].y;
      T     "coordinate".STAT118[1].STAT120;
_015: NOP   0;
      A     L 0.0;
      A(;
      L     "Timer".NumberVane;
      L     8;
      ==I;
      );
      =     L 0.1;
      A     L 0.1;
      JNB   _016;
      CALL  "BLKMOV" (
           SRCBLK                   := "DBWork".CoordSaldatura,
           RET_VAL                  := MW 2044,
           DSTBLK                   := "coordinate".STAT35);
_016: A     BR;
      R     "M75.1";
      A     L 0.1;
      JNB   _017;
      L     "DBWork".STAT29[1].x;
      T     "coordinate".STAT121[1].STAT122;
_017: NOP   0;
      A     L 0.1;
      JNB   _018;
      L     "DBWork".STAT29[1].y;
      T     "coordinate".STAT121[1].STAT123;
_018: NOP   0;
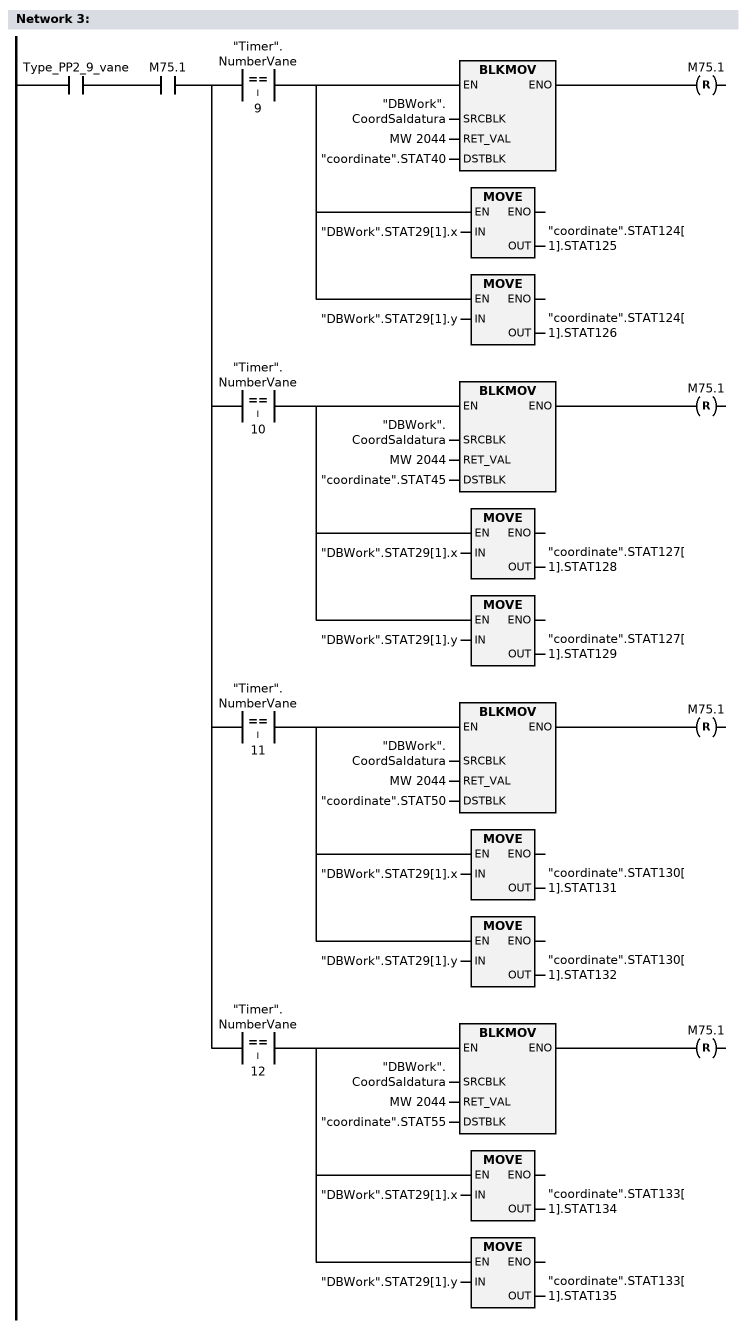
NETWORK
TITLE =
      A     "Type_PP2_9_vane";
      A     "M75.1";
      =     L 0.0;
      A     L 0.0;
      A(;
      L     "Timer".NumberVane;
      L     9;
      ==I;
      );
      =     L 0.1;
      A     L 0.1;
      JNB   _019;
      CALL  "BLKMOV" (
           SRCBLK                   := "DBWork".CoordSaldatura,
           RET_VAL                  := MW 2044,
           DSTBLK                   := "coordinate".STAT40);
_019: A     BR;
      R     "M75.1";
      A     L 0.1;
      JNB   _01a;
      L     "DBWork".STAT29[1].x;
      T     "coordinate".STAT124[1].STAT125;
_01a: NOP   0;
      A     L 0.1;
      JNB   _01b;
      L     "DBWork".STAT29[1].y;
      T     "coordinate".STAT124[1].STAT126;
_01b: NOP   0;
      A     L 0.0;
      A(;
      L     "Timer".NumberVane;
      L     10;
      ==I;
      );
      =     L 0.1;
      A     L 0.1;
      JNB   _01c;
      CALL  "BLKMOV" (
           SRCBLK                   := "DBWork".CoordSaldatura,
           RET_VAL                  := MW 2044,
           DSTBLK                   := "coordinate".STAT45);
_01c: A     BR;
      R     "M75.1";
      A     L 0.1;
      JNB   _01d;
      L     "DBWork".STAT29[1].x;
      T     "coordinate".STAT127[1].STAT128;
_01d: NOP   0;
      A     L 0.1;
      JNB   _01e;
      L     "DBWork".STAT29[1].y;
      T     "coordinate".STAT127[1].STAT129;
_01e: NOP   0;
      A     L 0.0;
      A(;
      L     "Timer".NumberVane;
      L     11;
      ==I;
      );
      =     L 0.1;
      A     L 0.1;
      JNB   _01f;
      CALL  "BLKMOV" (
           SRCBLK                   := "DBWork".CoordSaldatura,
           RET_VAL                  := MW 2044,
           DSTBLK                   := "coordinate".STAT50);
_01f: A     BR;
      R     "M75.1";
      A     L 0.1;
      JNB   _020;
      L     "DBWork".STAT29[1].x;
      T     "coordinate".STAT130[1].STAT131;
_020: NOP   0;
      A     L 0.1;
      JNB   _021;
      L     "DBWork".STAT29[1].y;
      T     "coordinate".STAT130[1].STAT132;
_021: NOP   0;
      A     L 0.0;
      A(;
      L     "Timer".NumberVane;
      L     12;
      ==I;
      );
      =     L 0.1;
      A     L 0.1;
      JNB   _022;
      CALL  "BLKMOV" (
           SRCBLK                   := "DBWork".CoordSaldatura,
           RET_VAL                  := MW 2044,
           DSTBLK                   := "coordinate".STAT55);
_022: A     BR;
      R     "M75.1";
      A     L 0.1;
      JNB   _023;
      L     "DBWork".STAT29[1].x;
      T     "coordinate".STAT133[1].STAT134;
_023: NOP   0;
      A     L 0.1;
      JNB   _024;
      L     "DBWork".STAT29[1].y;
      T     "coordinate".STAT133[1].STAT135;
_024: NOP   0;
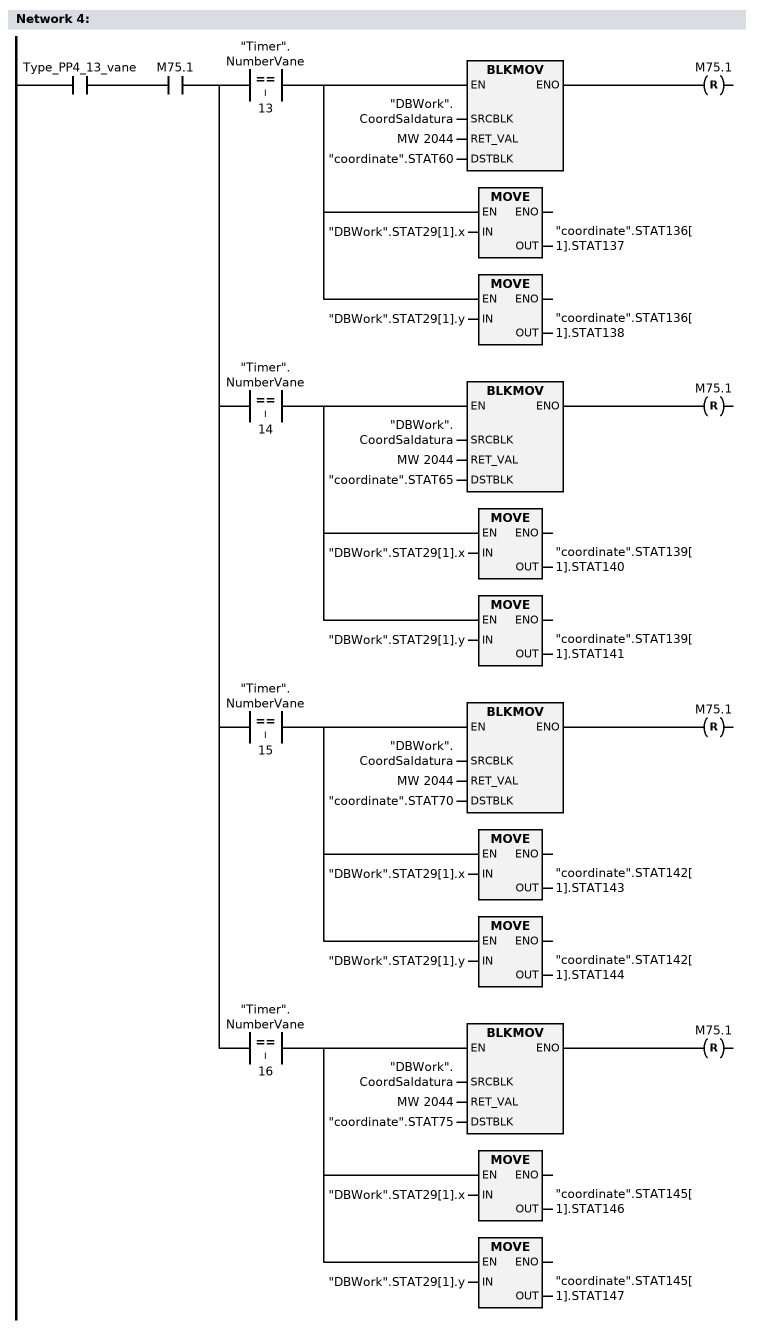
NETWORK
TITLE =
      A     "Type_PP4_13_vane";
      A     "M75.1";
      =     L 0.0;
      A     L 0.0;
      A(;
      L     "Timer".NumberVane;
      L     13;
      ==I;
      );
      =     L 0.1;
      A     L 0.1;
      JNB   _025;
      CALL  "BLKMOV" (
           SRCBLK                   := "DBWork".CoordSaldatura,
           RET_VAL                  := MW 2044,
           DSTBLK                   := "coordinate".STAT60);
_025: A     BR;
      R     "M75.1";
      A     L 0.1;
      JNB   _026;
      L     "DBWork".STAT29[1].x;
      T     "coordinate".STAT136[1].STAT137;
_026: NOP   0;
      A     L 0.1;
      JNB   _027;
      L     "DBWork".STAT29[1].y;
      T     "coordinate".STAT136[1].STAT138;
_027: NOP   0;
      A     L 0.0;
      A(;
      L     "Timer".NumberVane;
      L     14;
      ==I;
      );
      =     L 0.1;
      A     L 0.1;
      JNB   _028;
      CALL  "BLKMOV" (
           SRCBLK                   := "DBWork".CoordSaldatura,
           RET_VAL                  := MW 2044,
           DSTBLK                   := "coordinate".STAT65);
_028: A     BR;
      R     "M75.1";
      A     L 0.1;
      JNB   _029;
      L     "DBWork".STAT29[1].x;
      T     "coordinate".STAT139[1].STAT140;
_029: NOP   0;
      A     L 0.1;
      JNB   _02a;
      L     "DBWork".STAT29[1].y;
      T     "coordinate".STAT139[1].STAT141;
_02a: NOP   0;
      A     L 0.0;
      A(;
      L     "Timer".NumberVane;
      L     15;
      ==I;
      );
      =     L 0.1;
      A     L 0.1;
      JNB   _02b;
      CALL  "BLKMOV" (
           SRCBLK                   := "DBWork".CoordSaldatura,
           RET_VAL                  := MW 2044,
           DSTBLK                   := "coordinate".STAT70);
_02b: A     BR;
      R     "M75.1";
      A     L 0.1;
      JNB   _02c;
      L     "DBWork".STAT29[1].x;
      T     "coordinate".STAT142[1].STAT143;
_02c: NOP   0;
      A     L 0.1;
      JNB   _02d;
      L     "DBWork".STAT29[1].y;
      T     "coordinate".STAT142[1].STAT144;
_02d: NOP   0;
      A     L 0.0;
      A(;
      L     "Timer".NumberVane;
      L     16;
      ==I;
      );
      =     L 0.1;
      A     L 0.1;
      JNB   _02e;
      CALL  "BLKMOV" (
           SRCBLK                   := "DBWork".CoordSaldatura,
           RET_VAL                  := MW 2044,
           DSTBLK                   := "coordinate".STAT75);
_02e: A     BR;
      R     "M75.1";
      A     L 0.1;
      JNB   _02f;
      L     "DBWork".STAT29[1].x;
      T     "coordinate".STAT145[1].STAT146;
_02f: NOP   0;
      A     L 0.1;
      JNB   _030;
      L     "DBWork".STAT29[1].y;
      T     "coordinate".STAT145[1].STAT147;
_030: NOP   0;
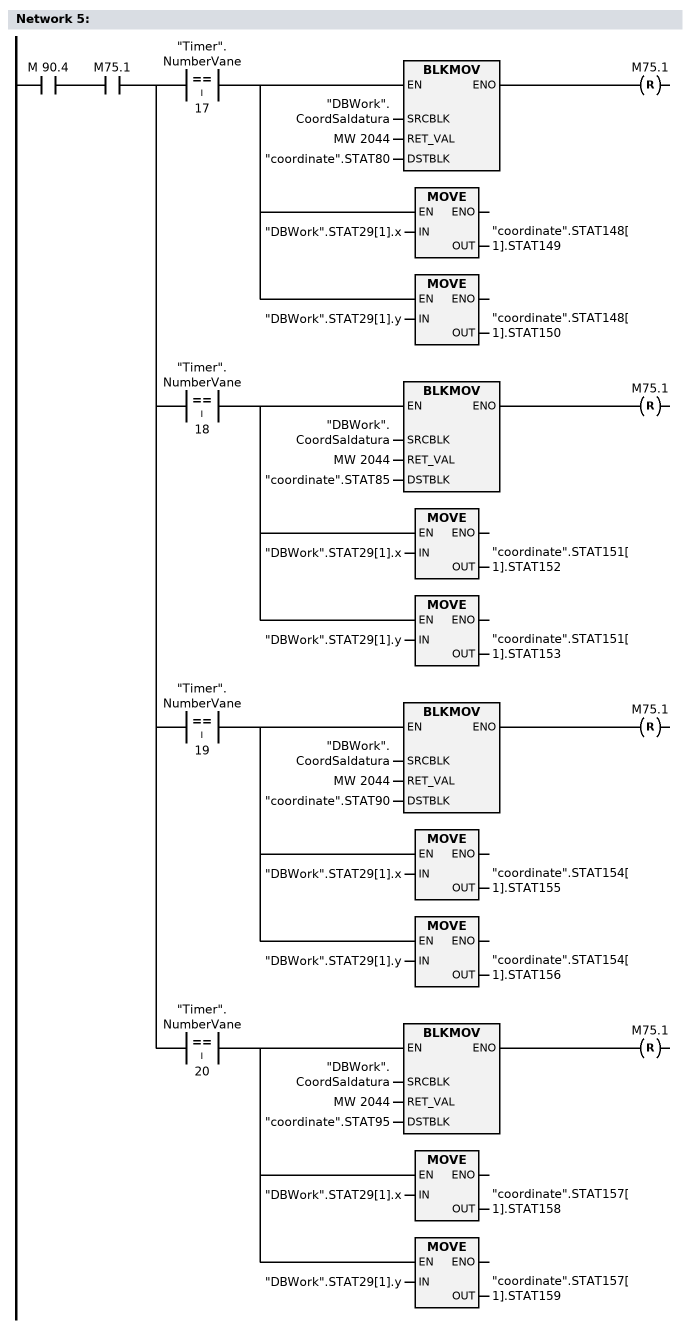
NETWORK
TITLE =
      A     M 90.4;
      A     "M75.1";
      =     L 0.0;
      A     L 0.0;
      A(;
      L     "Timer".NumberVane;
      L     17;
      ==I;
      );
      =     L 0.1;
      A     L 0.1;
      JNB   _031;
      CALL  "BLKMOV" (
           SRCBLK                   := "DBWork".CoordSaldatura,
           RET_VAL                  := MW 2044,
           DSTBLK                   := "coordinate".STAT80);
_031: A     BR;
      R     "M75.1";
      A     L 0.1;
      JNB   _032;
      L     "DBWork".STAT29[1].x;
      T     "coordinate".STAT148[1].STAT149;
_032: NOP   0;
      A     L 0.1;
      JNB   _033;
      L     "DBWork".STAT29[1].y;
      T     "coordinate".STAT148[1].STAT150;
_033: NOP   0;
      A     L 0.0;
      A(;
      L     "Timer".NumberVane;
      L     18;
      ==I;
      );
      =     L 0.1;
      A     L 0.1;
      JNB   _034;
      CALL  "BLKMOV" (
           SRCBLK                   := "DBWork".CoordSaldatura,
           RET_VAL                  := MW 2044,
           DSTBLK                   := "coordinate".STAT85);
_034: A     BR;
      R     "M75.1";
      A     L 0.1;
      JNB   _035;
      L     "DBWork".STAT29[1].x;
      T     "coordinate".STAT151[1].STAT152;
_035: NOP   0;
      A     L 0.1;
      JNB   _036;
      L     "DBWork".STAT29[1].y;
      T     "coordinate".STAT151[1].STAT153;
_036: NOP   0;
      A     L 0.0;
      A(;
      L     "Timer".NumberVane;
      L     19;
      ==I;
      );
      =     L 0.1;
      A     L 0.1;
      JNB   _037;
      CALL  "BLKMOV" (
           SRCBLK                   := "DBWork".CoordSaldatura,
           RET_VAL                  := MW 2044,
           DSTBLK                   := "coordinate".STAT90);
_037: A     BR;
      R     "M75.1";
      A     L 0.1;
      JNB   _038;
      L     "DBWork".STAT29[1].x;
      T     "coordinate".STAT154[1].STAT155;
_038: NOP   0;
      A     L 0.1;
      JNB   _039;
      L     "DBWork".STAT29[1].y;
      T     "coordinate".STAT154[1].STAT156;
_039: NOP   0;
      A     L 0.0;
      A(;
      L     "Timer".NumberVane;
      L     20;
      ==I;
      );
      =     L 0.1;
      A     L 0.1;
      JNB   _03a;
      CALL  "BLKMOV" (
           SRCBLK                   := "DBWork".CoordSaldatura,
           RET_VAL                  := MW 2044,
           DSTBLK                   := "coordinate".STAT95);
_03a: A     BR;
      R     "M75.1";
      A     L 0.1;
      JNB   _03b;
      L     "DBWork".STAT29[1].x;
      T     "coordinate".STAT157[1].STAT158;
_03b: NOP   0;
      A     L 0.1;
      JNB   _03c;
      L     "DBWork".STAT29[1].y;
      T     "coordinate".STAT157[1].STAT159;
_03c: NOP   0;
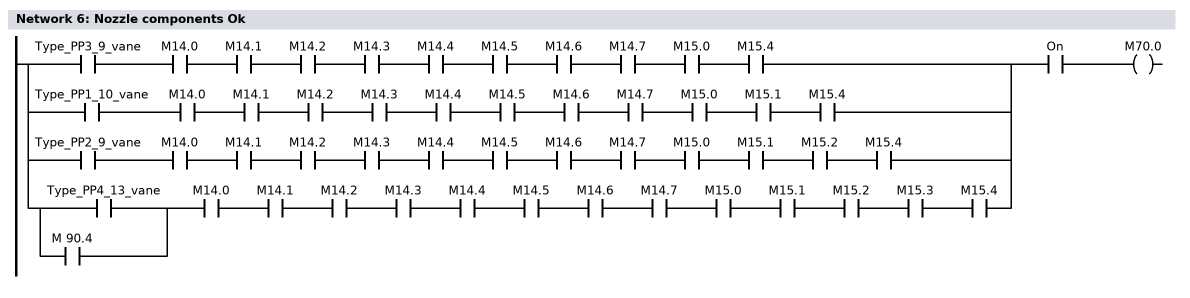
NETWORK
TITLE = Nozzle components Ok
      A(;
      A     "Type_PP3_9_vane";
      A     "M14.0";
      A     "M14.1";
      A     "M14.2";
      A     "M14.3";
      A     "M14.4";
      A     "M14.5";
      A     "M14.6";
      A     "M14.7";
      A     "M15.0";
      A     "M15.4";
      O;
      A     "Type_PP1_10_vane";
      A     "M14.0";
      A     "M14.1";
      A     "M14.2";
      A     "M14.3";
      A     "M14.4";
      A     "M14.5";
      A     "M14.6";
      A     "M14.7";
      A     "M15.0";
      A     "M15.1";
      A     "M15.4";
      O;
      A     "Type_PP2_9_vane";
      A     "M14.0";
      A     "M14.1";
      A     "M14.2";
      A     "M14.3";
      A     "M14.4";
      A     "M14.5";
      A     "M14.6";
      A     "M14.7";
      A     "M15.0";
      A     "M15.1";
      A     "M15.2";
      A     "M15.4";
      O;
      A(;
      O     "Type_PP4_13_vane";
      O     M 90.4;
      );
      A     "M14.0";
      A     "M14.1";
      A     "M14.2";
      A     "M14.3";
      A     "M14.4";
      A     "M14.5";
      A     "M14.6";
      A     "M14.7";
      A     "M15.0";
      A     "M15.1";
      A     "M15.2";
      A     "M15.3";
      A     "M15.4";
      );
      A     "On";
      =     "M70.0";
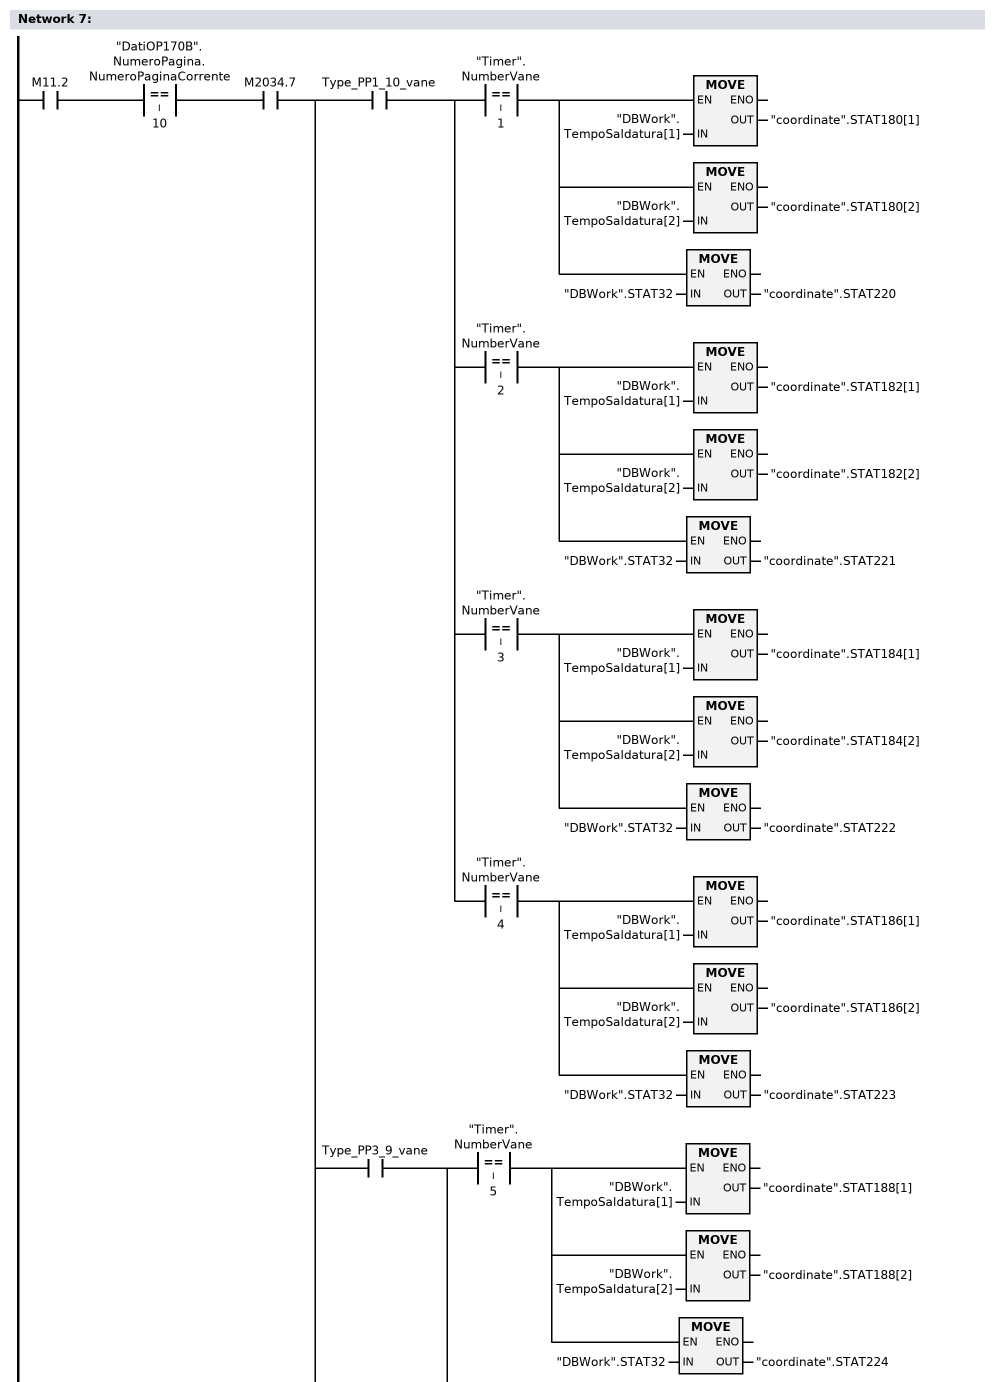
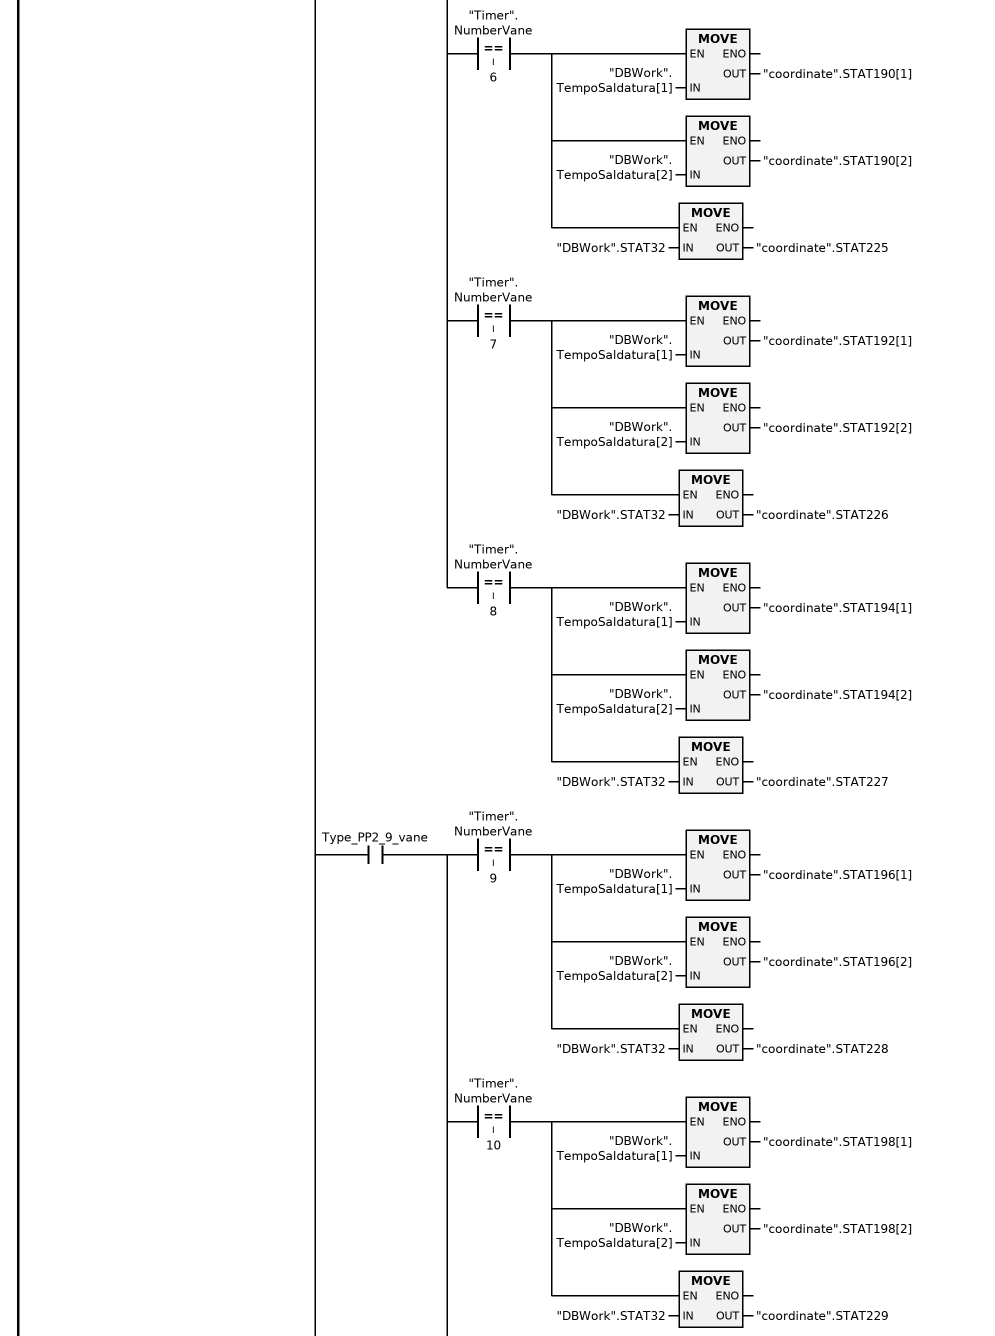
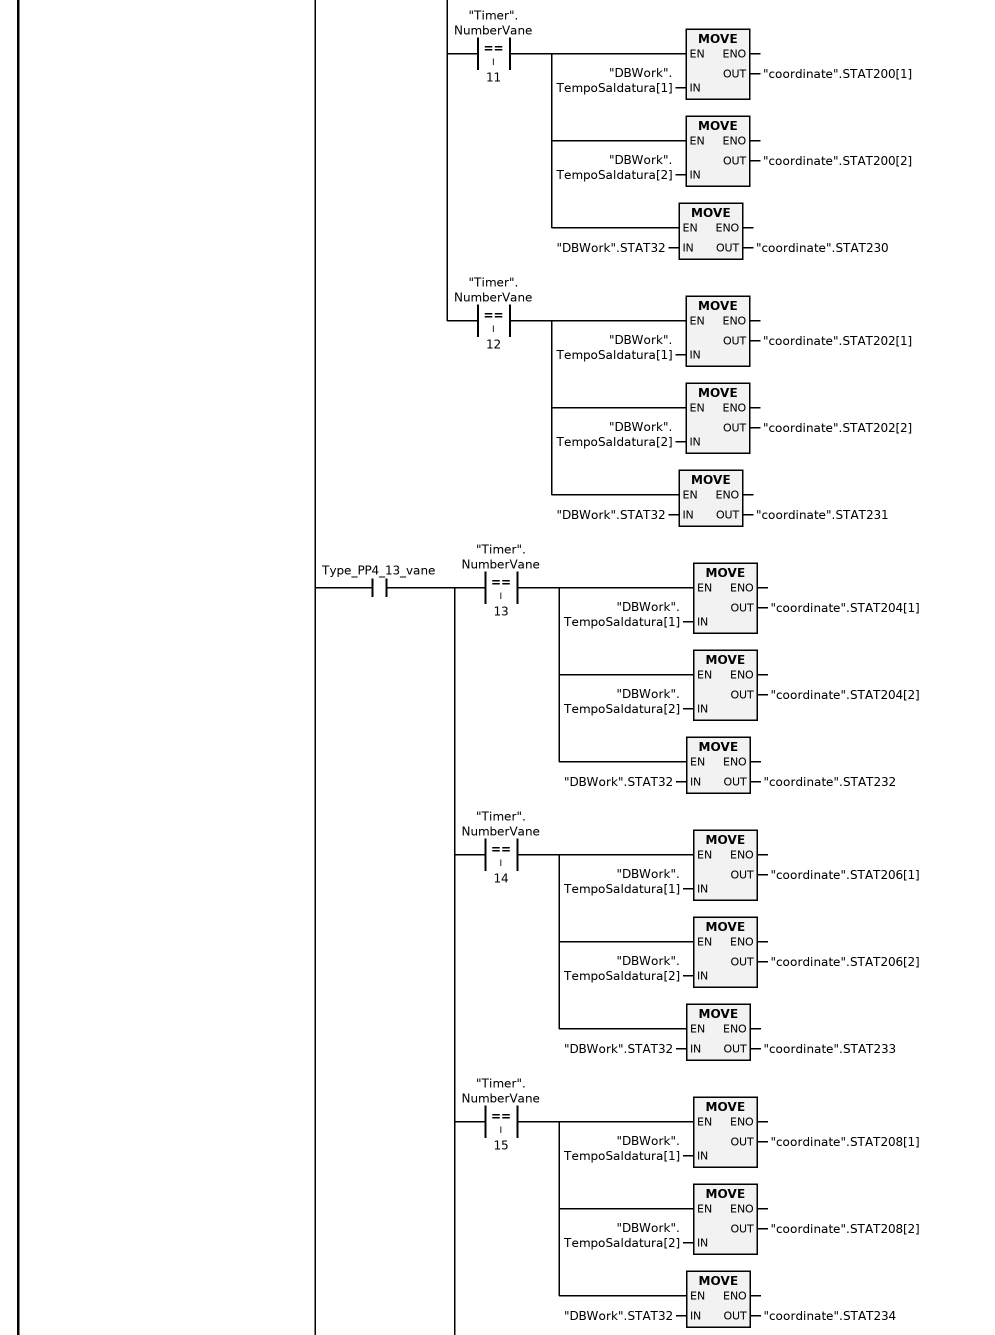
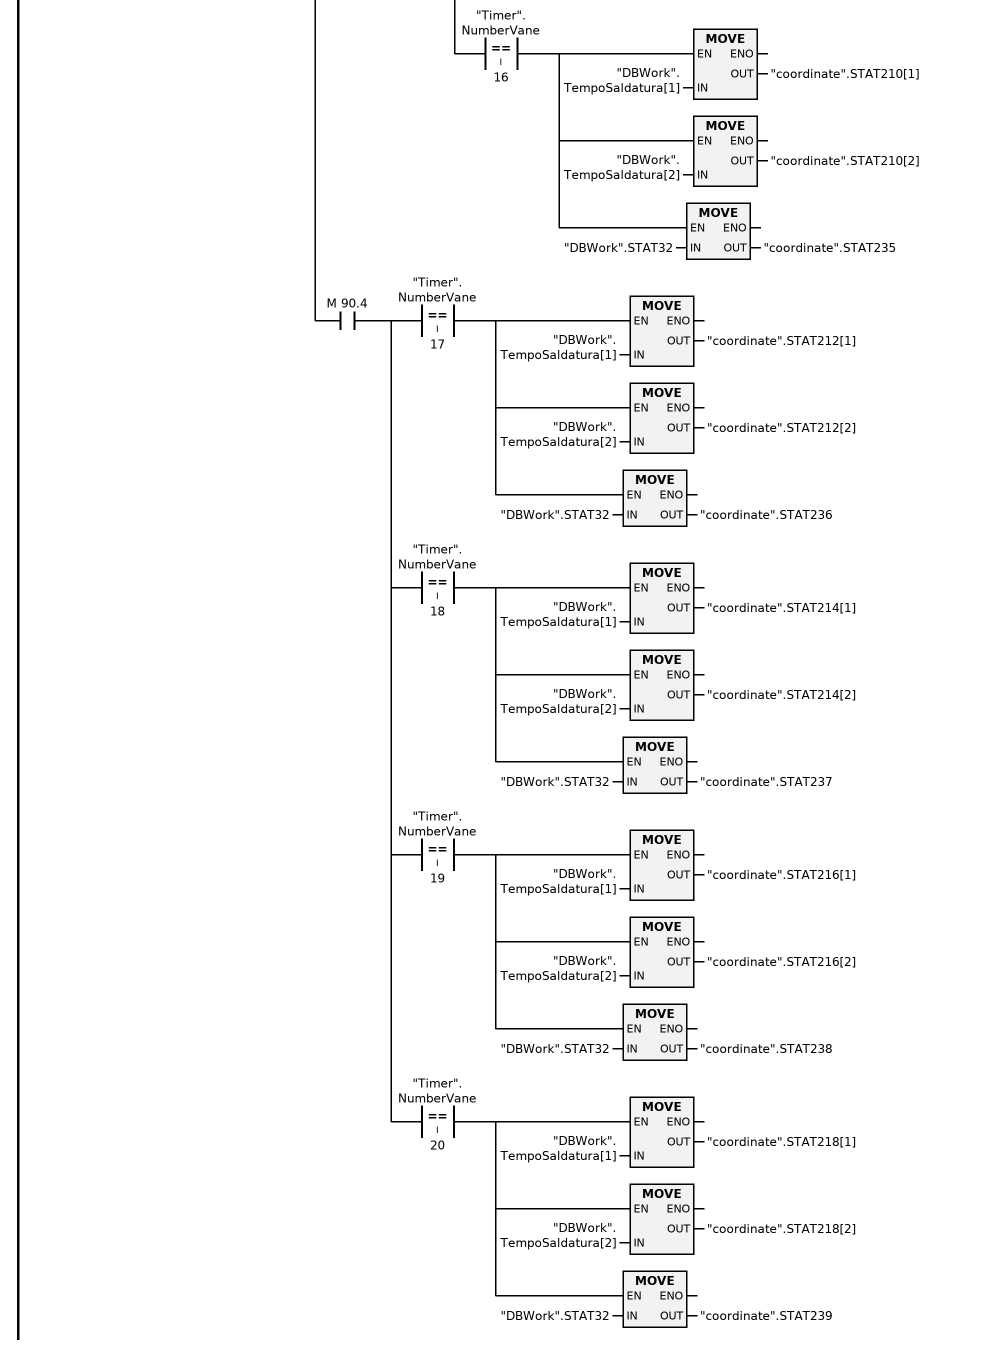
NETWORK
TITLE =
      A     "M11.2";
      A(;
      L     "DatiOP170B".NumeroPagina.NumeroPaginaCorrente;
      L     10;
      ==I;
      );
      A     "M2034.7";
      =     L 0.0;
      A     L 0.0;
      A     "Type_PP1_10_vane";
      =     L 0.1;
      A     L 0.1;
      A(;
      L     "Timer".NumberVane;
      L     1;
      ==I;
      );
      =     L 0.2;
      A     L 0.2;
      JNB   _03d;
      L     "DBWork".TempoSaldatura[1];
      T     "coordinate".STAT180[1];
_03d: NOP   0;
      A     L 0.2;
      JNB   _03e;
      L     "DBWork".TempoSaldatura[2];
      T     "coordinate".STAT180[2];
_03e: NOP   0;
      A     L 0.2;
      JNB   _03f;
      L     "DBWork".STAT32;
      T     "coordinate".STAT220;
_03f: NOP   0;
      A     L 0.1;
      A(;
      L     "Timer".NumberVane;
      L     2;
      ==I;
      );
      =     L 0.2;
      A     L 0.2;
      JNB   _040;
      L     "DBWork".TempoSaldatura[1];
      T     "coordinate".STAT182[1];
_040: NOP   0;
      A     L 0.2;
      JNB   _041;
      L     "DBWork".TempoSaldatura[2];
      T     "coordinate".STAT182[2];
_041: NOP   0;
      A     L 0.2;
      JNB   _042;
      L     "DBWork".STAT32;
      T     "coordinate".STAT221;
_042: NOP   0;
      A     L 0.1;
      A(;
      L     "Timer".NumberVane;
      L     3;
      ==I;
      );
      =     L 0.2;
      A     L 0.2;
      JNB   _043;
      L     "DBWork".TempoSaldatura[1];
      T     "coordinate".STAT184[1];
_043: NOP   0;
      A     L 0.2;
      JNB   _044;
      L     "DBWork".TempoSaldatura[2];
      T     "coordinate".STAT184[2];
_044: NOP   0;
      A     L 0.2;
      JNB   _045;
      L     "DBWork".STAT32;
      T     "coordinate".STAT222;
_045: NOP   0;
      A     L 0.1;
      A(;
      L     "Timer".NumberVane;
      L     4;
      ==I;
      );
      =     L 0.2;
      A     L 0.2;
      JNB   _046;
      L     "DBWork".TempoSaldatura[1];
      T     "coordinate".STAT186[1];
_046: NOP   0;
      A     L 0.2;
      JNB   _047;
      L     "DBWork".TempoSaldatura[2];
      T     "coordinate".STAT186[2];
_047: NOP   0;
      A     L 0.2;
      JNB   _048;
      L     "DBWork".STAT32;
      T     "coordinate".STAT223;
_048: NOP   0;
      A     L 0.0;
      A     "Type_PP3_9_vane";
      =     L 0.1;
      A     L 0.1;
      A(;
      L     "Timer".NumberVane;
      L     5;
      ==I;
      );
      =     L 0.2;
      A     L 0.2;
      JNB   _049;
      L     "DBWork".TempoSaldatura[1];
      T     "coordinate".STAT188[1];
_049: NOP   0;
      A     L 0.2;
      JNB   _04a;
      L     "DBWork".TempoSaldatura[2];
      T     "coordinate".STAT188[2];
_04a: NOP   0;
      A     L 0.2;
      JNB   _04b;
      L     "DBWork".STAT32;
      T     "coordinate".STAT224;
_04b: NOP   0;
      A     L 0.1;
      A(;
      L     "Timer".NumberVane;
      L     6;
      ==I;
      );
      =     L 0.2;
      A     L 0.2;
      JNB   _04c;
      L     "DBWork".TempoSaldatura[1];
      T     "coordinate".STAT190[1];
_04c: NOP   0;
      A     L 0.2;
      JNB   _04d;
      L     "DBWork".TempoSaldatura[2];
      T     "coordinate".STAT190[2];
_04d: NOP   0;
      A     L 0.2;
      JNB   _04e;
      L     "DBWork".STAT32;
      T     "coordinate".STAT225;
_04e: NOP   0;
      A     L 0.1;
      A(;
      L     "Timer".NumberVane;
      L     7;
      ==I;
      );
      =     L 0.2;
      A     L 0.2;
      JNB   _04f;
      L     "DBWork".TempoSaldatura[1];
      T     "coordinate".STAT192[1];
_04f: NOP   0;
      A     L 0.2;
      JNB   _050;
      L     "DBWork".TempoSaldatura[2];
      T     "coordinate".STAT192[2];
_050: NOP   0;
      A     L 0.2;
      JNB   _051;
      L     "DBWork".STAT32;
      T     "coordinate".STAT226;
_051: NOP   0;
      A     L 0.1;
      A(;
      L     "Timer".NumberVane;
      L     8;
      ==I;
      );
      =     L 0.2;
      A     L 0.2;
      JNB   _052;
      L     "DBWork".TempoSaldatura[1];
      T     "coordinate".STAT194[1];
_052: NOP   0;
      A     L 0.2;
      JNB   _053;
      L     "DBWork".TempoSaldatura[2];
      T     "coordinate".STAT194[2];
_053: NOP   0;
      A     L 0.2;
      JNB   _054;
      L     "DBWork".STAT32;
      T     "coordinate".STAT227;
_054: NOP   0;
      A     L 0.0;
      A     "Type_PP2_9_vane";
      =     L 0.1;
      A     L 0.1;
      A(;
      L     "Timer".NumberVane;
      L     9;
      ==I;
      );
      =     L 0.2;
      A     L 0.2;
      JNB   _055;
      L     "DBWork".TempoSaldatura[1];
      T     "coordinate".STAT196[1];
_055: NOP   0;
      A     L 0.2;
      JNB   _056;
      L     "DBWork".TempoSaldatura[2];
      T     "coordinate".STAT196[2];
_056: NOP   0;
      A     L 0.2;
      JNB   _057;
      L     "DBWork".STAT32;
      T     "coordinate".STAT228;
_057: NOP   0;
      A     L 0.1;
      A(;
      L     "Timer".NumberVane;
      L     10;
      ==I;
      );
      =     L 0.2;
      A     L 0.2;
      JNB   _058;
      L     "DBWork".TempoSaldatura[1];
      T     "coordinate".STAT198[1];
_058: NOP   0;
      A     L 0.2;
      JNB   _059;
      L     "DBWork".TempoSaldatura[2];
      T     "coordinate".STAT198[2];
_059: NOP   0;
      A     L 0.2;
      JNB   _05a;
      L     "DBWork".STAT32;
      T     "coordinate".STAT229;
_05a: NOP   0;
      A     L 0.1;
      A(;
      L     "Timer".NumberVane;
      L     11;
      ==I;
      );
      =     L 0.2;
      A     L 0.2;
      JNB   _05b;
      L     "DBWork".TempoSaldatura[1];
      T     "coordinate".STAT200[1];
_05b: NOP   0;
      A     L 0.2;
      JNB   _05c;
      L     "DBWork".TempoSaldatura[2];
      T     "coordinate".STAT200[2];
_05c: NOP   0;
      A     L 0.2;
      JNB   _05d;
      L     "DBWork".STAT32;
      T     "coordinate".STAT230;
_05d: NOP   0;
      A     L 0.1;
      A(;
      L     "Timer".NumberVane;
      L     12;
      ==I;
      );
      =     L 0.2;
      A     L 0.2;
      JNB   _05e;
      L     "DBWork".TempoSaldatura[1];
      T     "coordinate".STAT202[1];
_05e: NOP   0;
      A     L 0.2;
      JNB   _05f;
      L     "DBWork".TempoSaldatura[2];
      T     "coordinate".STAT202[2];
_05f: NOP   0;
      A     L 0.2;
      JNB   _060;
      L     "DBWork".STAT32;
      T     "coordinate".STAT231;
_060: NOP   0;
      A     L 0.0;
      A     "Type_PP4_13_vane";
      =     L 0.1;
      A     L 0.1;
      A(;
      L     "Timer".NumberVane;
      L     13;
      ==I;
      );
      =     L 0.2;
      A     L 0.2;
      JNB   _061;
      L     "DBWork".TempoSaldatura[1];
      T     "coordinate".STAT204[1];
_061: NOP   0;
      A     L 0.2;
      JNB   _062;
      L     "DBWork".TempoSaldatura[2];
      T     "coordinate".STAT204[2];
_062: NOP   0;
      A     L 0.2;
      JNB   _063;
      L     "DBWork".STAT32;
      T     "coordinate".STAT232;
_063: NOP   0;
      A     L 0.1;
      A(;
      L     "Timer".NumberVane;
      L     14;
      ==I;
      );
      =     L 0.2;
      A     L 0.2;
      JNB   _064;
      L     "DBWork".TempoSaldatura[1];
      T     "coordinate".STAT206[1];
_064: NOP   0;
      A     L 0.2;
      JNB   _065;
      L     "DBWork".TempoSaldatura[2];
      T     "coordinate".STAT206[2];
_065: NOP   0;
      A     L 0.2;
      JNB   _066;
      L     "DBWork".STAT32;
      T     "coordinate".STAT233;
_066: NOP   0;
      A     L 0.1;
      A(;
      L     "Timer".NumberVane;
      L     15;
      ==I;
      );
      =     L 0.2;
      A     L 0.2;
      JNB   _067;
      L     "DBWork".TempoSaldatura[1];
      T     "coordinate".STAT208[1];
_067: NOP   0;
      A     L 0.2;
      JNB   _068;
      L     "DBWork".TempoSaldatura[2];
      T     "coordinate".STAT208[2];
_068: NOP   0;
      A     L 0.2;
      JNB   _069;
      L     "DBWork".STAT32;
      T     "coordinate".STAT234;
_069: NOP   0;
      A     L 0.1;
      A(;
      L     "Timer".NumberVane;
      L     16;
      ==I;
      );
      =     L 0.2;
      A     L 0.2;
      JNB   _06a;
      L     "DBWork".TempoSaldatura[1];
      T     "coordinate".STAT210[1];
_06a: NOP   0;
      A     L 0.2;
      JNB   _06b;
      L     "DBWork".TempoSaldatura[2];
      T     "coordinate".STAT210[2];
_06b: NOP   0;
      A     L 0.2;
      JNB   _06c;
      L     "DBWork".STAT32;
      T     "coordinate".STAT235;
_06c: NOP   0;
      A     L 0.0;
      A     M 90.4;
      =     L 0.1;
      A     L 0.1;
      A(;
      L     "Timer".NumberVane;
      L     17;
      ==I;
      );
      =     L 0.2;
      A     L 0.2;
      JNB   _06d;
      L     "DBWork".TempoSaldatura[1];
      T     "coordinate".STAT212[1];
_06d: NOP   0;
      A     L 0.2;
      JNB   _06e;
      L     "DBWork".TempoSaldatura[2];
      T     "coordinate".STAT212[2];
_06e: NOP   0;
      A     L 0.2;
      JNB   _06f;
      L     "DBWork".STAT32;
      T     "coordinate".STAT236;
_06f: NOP   0;
      A     L 0.1;
      A(;
      L     "Timer".NumberVane;
      L     18;
      ==I;
      );
      =     L 0.2;
      A     L 0.2;
      JNB   _070;
      L     "DBWork".TempoSaldatura[1];
      T     "coordinate".STAT214[1];
_070: NOP   0;
      A     L 0.2;
      JNB   _071;
      L     "DBWork".TempoSaldatura[2];
      T     "coordinate".STAT214[2];
_071: NOP   0;
      A     L 0.2;
      JNB   _072;
      L     "DBWork".STAT32;
      T     "coordinate".STAT237;
_072: NOP   0;
      A     L 0.1;
      A(;
      L     "Timer".NumberVane;
      L     19;
      ==I;
      );
      =     L 0.2;
      A     L 0.2;
      JNB   _073;
      L     "DBWork".TempoSaldatura[1];
      T     "coordinate".STAT216[1];
_073: NOP   0;
      A     L 0.2;
      JNB   _074;
      L     "DBWork".TempoSaldatura[2];
      T     "coordinate".STAT216[2];
_074: NOP   0;
      A     L 0.2;
      JNB   _075;
      L     "DBWork".STAT32;
      T     "coordinate".STAT238;
_075: NOP   0;
      A     L 0.1;
      A(;
      L     "Timer".NumberVane;
      L     20;
      ==I;
      );
      =     L 0.2;
      A     L 0.2;
      JNB   _076;
      L     "DBWork".TempoSaldatura[1];
      T     "coordinate".STAT218[1];
_076: NOP   0;
      A     L 0.2;
      JNB   _077;
      L     "DBWork".TempoSaldatura[2];
      T     "coordinate".STAT218[2];
_077: NOP   0;
      A     L 0.2;
      JNB   _078;
      L     "DBWork".STAT32;
      T     "coordinate".STAT239;
_078: NOP   0;
NETWORK
TITLE =
NETWORK
TITLE =
      A     "On";
      =     L 0.0;
      A     L 0.0;
      A(;
      A(;
      L     "DBWork".PP[1].NumSaldaturaAtt;
      L     0;
      ==I;
      );
      A     "AUT";
      O;
      A     "M11.2";
      A(;
      L     "DatiOP170B".PointWeldingTeachIn;
      L     1;
      ==I;
      );
      A(;
      O(;
      L     "DatiOP170B".NumeroPagina.NumeroPaginaCorrente;
      L     5;
      ==I;
      );
      O(;
      L     "DatiOP170B".NumeroPagina.NumeroPaginaCorrente;
      L     11;
      ==I;
      );
      );
      );
      =     L 0.1;
      A(;
      A     L 0.1;
      A     "DBWork".RotationTable;
      JNB   _079;
      L     "DBWork".CoordSaldatura[1].X1;
      T     "MD588";
      SET;
      SAVE;
      CLR;
_079: A     BR;
      );
      JNB   _07a;
      L     "DBWork".CoordSaldatura[1].Y1;
      T     "MD592";
_07a: NOP   0;
      A(;
      A     L 0.1;
      AN    "DBWork".RotationTable;
      JNB   _07b;
      L     "DBWork".CoordSaldatura[1].X2;
      T     "MD588";
      SET;
      SAVE;
      CLR;
_07b: A     BR;
      );
      JNB   _07c;
      L     "DBWork".CoordSaldatura[1].Y2;
      T     "MD592";
_07c: NOP   0;
      A     L 0.0;
      A(;
      A(;
      L     "DBWork".PP[1].NumSaldaturaAtt;
      L     1;
      ==I;
      );
      A     "AUT";
      O;
      A     "M11.2";
      A(;
      L     "DatiOP170B".PointWeldingTeachIn;
      L     2;
      ==I;
      );
      A(;
      O(;
      L     "DatiOP170B".NumeroPagina.NumeroPaginaCorrente;
      L     5;
      ==I;
      );
      O(;
      L     "DatiOP170B".NumeroPagina.NumeroPaginaCorrente;
      L     11;
      ==I;
      );
      );
      );
      =     L 0.1;
      A(;
      A     L 0.1;
      A     "DBWork".RotationTable;
      JNB   _07d;
      L     "DBWork".CoordSaldatura[2].X1;
      T     "MD588";
      SET;
      SAVE;
      CLR;
_07d: A     BR;
      );
      JNB   _07e;
      L     "DBWork".CoordSaldatura[2].Y1;
      T     "MD592";
_07e: NOP   0;
      A(;
      A     L 0.1;
      AN    "DBWork".RotationTable;
      JNB   _07f;
      L     "DBWork".CoordSaldatura[2].X2;
      T     "MD588";
      SET;
      SAVE;
      CLR;
_07f: A     BR;
      );
      JNB   _080;
      L     "DBWork".CoordSaldatura[2].Y2;
      T     "MD592";
_080: NOP   0;
      A     L 0.0;
      A(;
      A(;
      L     "DBWork".PP[1].NumSaldaturaAtt;
      L     2;
      ==I;
      );
      A     "AUT";
      O;
      A     "M11.2";
      A(;
      L     "DatiOP170B".PointWeldingTeachIn;
      L     3;
      ==I;
      );
      A(;
      O(;
      L     "DatiOP170B".NumeroPagina.NumeroPaginaCorrente;
      L     5;
      ==I;
      );
      O(;
      L     "DatiOP170B".NumeroPagina.NumeroPaginaCorrente;
      L     11;
      ==I;
      );
      );
      );
      =     L 0.1;
      A(;
      A     L 0.1;
      A     "DBWork".RotationTable;
      JNB   _081;
      L     "DBWork".CoordSaldatura[3].X1;
      T     "MD588";
      SET;
      SAVE;
      CLR;
_081: A     BR;
      );
      JNB   _082;
      L     "DBWork".CoordSaldatura[3].Y1;
      T     "MD592";
_082: NOP   0;
      A(;
      A     L 0.1;
      AN    "DBWork".RotationTable;
      JNB   _083;
      L     "DBWork".CoordSaldatura[3].X2;
      T     "MD588";
      SET;
      SAVE;
      CLR;
_083: A     BR;
      );
      JNB   _084;
      L     "DBWork".CoordSaldatura[3].Y2;
      T     "MD592";
_084: NOP   0;
      A     L 0.0;
      A(;
      A(;
      L     "DBWork".PP[1].NumSaldaturaAtt;
      L     3;
      ==I;
      );
      A     "AUT";
      O;
      A     "M11.2";
      A(;
      L     "DatiOP170B".PointWeldingTeachIn;
      L     4;
      ==I;
      );
      A(;
      O(;
      L     "DatiOP170B".NumeroPagina.NumeroPaginaCorrente;
      L     5;
      ==I;
      );
      O(;
      L     "DatiOP170B".NumeroPagina.NumeroPaginaCorrente;
      L     11;
      ==I;
      );
      );
      );
      =     L 0.1;
      A(;
      A     L 0.1;
      A     "DBWork".RotationTable;
      JNB   _085;
      L     "DBWork".CoordSaldatura[4].X1;
      T     "MD588";
      SET;
      SAVE;
      CLR;
_085: A     BR;
      );
      JNB   _086;
      L     "DBWork".CoordSaldatura[4].Y1;
      T     "MD592";
_086: NOP   0;
      A(;
      A     L 0.1;
      AN    "DBWork".RotationTable;
      JNB   _087;
      L     "DBWork".CoordSaldatura[4].X2;
      T     "MD588";
      SET;
      SAVE;
      CLR;
_087: A     BR;
      );
      JNB   _088;
      L     "DBWork".CoordSaldatura[4].Y2;
      T     "MD592";
_088: NOP   0;
      A     L 0.0;
      A(;
      A(;
      L     "DBWork".PP[1].NumSaldaturaAtt;
      L     4;
      ==I;
      );
      A     "AUT";
      O;
      A     "M11.2";
      A(;
      L     "DatiOP170B".PointWeldingTeachIn;
      L     5;
      ==I;
      );
      A(;
      O(;
      L     "DatiOP170B".NumeroPagina.NumeroPaginaCorrente;
      L     5;
      ==I;
      );
      O(;
      L     "DatiOP170B".NumeroPagina.NumeroPaginaCorrente;
      L     11;
      ==I;
      );
      );
      );
      =     L 0.1;
      A(;
      A     L 0.1;
      A     "DBWork".RotationTable;
      JNB   _089;
      L     "DBWork".CoordSaldatura[5].X1;
      T     "MD588";
      SET;
      SAVE;
      CLR;
_089: A     BR;
      );
      JNB   _08a;
      L     "DBWork".CoordSaldatura[5].Y1;
      T     "MD592";
_08a: NOP   0;
      A(;
      A     L 0.1;
      AN    "DBWork".RotationTable;
      JNB   _08b;
      L     "DBWork".CoordSaldatura[5].X2;
      T     "MD588";
      SET;
      SAVE;
      CLR;
_08b: A     BR;
      );
      JNB   _08c;
      L     "DBWork".CoordSaldatura[5].Y2;
      T     "MD592";
_08c: NOP   0;
      A     L 0.0;
      A(;
      A(;
      L     "DBWork".PP[1].NumSaldaturaAtt;
      L     5;
      ==I;
      );
      A     "AUT";
      O;
      A     "M11.2";
      A(;
      L     "DatiOP170B".PointWeldingTeachIn;
      L     6;
      ==I;
      );
      A(;
      O(;
      L     "DatiOP170B".NumeroPagina.NumeroPaginaCorrente;
      L     5;
      ==I;
      );
      O(;
      L     "DatiOP170B".NumeroPagina.NumeroPaginaCorrente;
      L     11;
      ==I;
      );
      );
      );
      =     L 0.1;
      A(;
      A     L 0.1;
      A     "DBWork".RotationTable;
      JNB   _08d;
      L     "DBWork".CoordSaldatura[6].X1;
      T     "MD588";
      SET;
      SAVE;
      CLR;
_08d: A     BR;
      );
      JNB   _08e;
      L     "DBWork".CoordSaldatura[6].Y1;
      T     "MD592";
_08e: NOP   0;
      A(;
      A     L 0.1;
      AN    "DBWork".RotationTable;
      JNB   _08f;
      L     "DBWork".CoordSaldatura[6].X2;
      T     "MD588";
      SET;
      SAVE;
      CLR;
_08f: A     BR;
      );
      JNB   _090;
      L     "DBWork".CoordSaldatura[6].Y2;
      T     "MD592";
_090: NOP   0;
      A     L 0.0;
      A(;
      A(;
      L     "DBWork".PP[1].NumSaldaturaAtt;
      L     6;
      ==I;
      );
      A     "AUT";
      O;
      A     "M11.2";
      A(;
      L     "DatiOP170B".PointWeldingTeachIn;
      L     7;
      ==I;
      );
      A(;
      O(;
      L     "DatiOP170B".NumeroPagina.NumeroPaginaCorrente;
      L     5;
      ==I;
      );
      O(;
      L     "DatiOP170B".NumeroPagina.NumeroPaginaCorrente;
      L     11;
      ==I;
      );
      );
      );
      =     L 0.1;
      A(;
      A     L 0.1;
      A     "DBWork".RotationTable;
      JNB   _091;
      L     "DBWork".CoordSaldatura[7].X1;
      T     "MD588";
      SET;
      SAVE;
      CLR;
_091: A     BR;
      );
      JNB   _092;
      L     "DBWork".CoordSaldatura[7].Y1;
      T     "MD592";
_092: NOP   0;
      A(;
      A     L 0.1;
      AN    "DBWork".RotationTable;
      JNB   _093;
      L     "DBWork".CoordSaldatura[7].X2;
      T     "MD588";
      SET;
      SAVE;
      CLR;
_093: A     BR;
      );
      JNB   _094;
      L     "DBWork".CoordSaldatura[7].Y2;
      T     "MD592";
_094: NOP   0;
      A     L 0.0;
      A(;
      A(;
      L     "DBWork".PP[1].NumSaldaturaAtt;
      L     7;
      ==I;
      );
      A     "AUT";
      O;
      A     "M11.2";
      A(;
      L     "DatiOP170B".PointWeldingTeachIn;
      L     8;
      ==I;
      );
      A(;
      O(;
      L     "DatiOP170B".NumeroPagina.NumeroPaginaCorrente;
      L     5;
      ==I;
      );
      O(;
      L     "DatiOP170B".NumeroPagina.NumeroPaginaCorrente;
      L     11;
      ==I;
      );
      );
      );
      =     L 0.1;
      A(;
      A     L 0.1;
      A     "DBWork".RotationTable;
      JNB   _095;
      L     "DBWork".CoordSaldatura[8].X1;
      T     "MD588";
      SET;
      SAVE;
      CLR;
_095: A     BR;
      );
      JNB   _096;
      L     "DBWork".CoordSaldatura[8].Y1;
      T     "MD592";
_096: NOP   0;
      A(;
      A     L 0.1;
      AN    "DBWork".RotationTable;
      JNB   _097;
      L     "DBWork".CoordSaldatura[8].X2;
      T     "MD588";
      SET;
      SAVE;
      CLR;
_097: A     BR;
      );
      JNB   _098;
      L     "DBWork".CoordSaldatura[8].Y2;
      T     "MD592";
_098: NOP   0;
      A     L 0.0;
      A(;
      A(;
      L     "DBWork".PP[1].NumSaldaturaAtt;
      L     8;
      ==I;
      );
      A     "AUT";
      O;
      A     "M11.2";
      A(;
      L     "DatiOP170B".PointWeldingTeachIn;
      L     9;
      ==I;
      );
      A(;
      O(;
      L     "DatiOP170B".NumeroPagina.NumeroPaginaCorrente;
      L     5;
      ==I;
      );
      O(;
      L     "DatiOP170B".NumeroPagina.NumeroPaginaCorrente;
      L     11;
      ==I;
      );
      );
      );
      =     L 0.1;
      A(;
      A     L 0.1;
      A     "DBWork".RotationTable;
      JNB   _099;
      L     "DBWork".CoordSaldatura[9].X1;
      T     "MD588";
      SET;
      SAVE;
      CLR;
_099: A     BR;
      );
      JNB   _09a;
      L     "DBWork".CoordSaldatura[9].Y1;
      T     "MD592";
_09a: NOP   0;
      A(;
      A     L 0.1;
      AN    "DBWork".RotationTable;
      JNB   _09b;
      L     "DBWork".CoordSaldatura[9].X2;
      T     "MD588";
      SET;
      SAVE;
      CLR;
_09b: A     BR;
      );
      JNB   _09c;
      L     "DBWork".CoordSaldatura[9].Y2;
      T     "MD592";
_09c: NOP   0;
      A     L 0.0;
      A(;
      A(;
      L     "DBWork".PP[1].NumSaldaturaAtt;
      L     9;
      ==I;
      );
      A     "AUT";
      O;
      A     "M11.2";
      A(;
      L     "DatiOP170B".PointWeldingTeachIn;
      L     10;
      ==I;
      );
      A(;
      O(;
      L     "DatiOP170B".NumeroPagina.NumeroPaginaCorrente;
      L     5;
      ==I;
      );
      O(;
      L     "DatiOP170B".NumeroPagina.NumeroPaginaCorrente;
      L     11;
      ==I;
      );
      );
      );
      =     L 0.1;
      A(;
      A     L 0.1;
      A     "DBWork".RotationTable;
      JNB   _09d;
      L     "DBWork".CoordSaldatura[10].X1;
      T     "MD588";
      SET;
      SAVE;
      CLR;
_09d: A     BR;
      );
      JNB   _09e;
      L     "DBWork".CoordSaldatura[10].Y1;
      T     "MD592";
_09e: NOP   0;
      A(;
      A     L 0.1;
      AN    "DBWork".RotationTable;
      JNB   _09f;
      L     "DBWork".CoordSaldatura[10].X2;
      T     "MD588";
      SET;
      SAVE;
      CLR;
_09f: A     BR;
      );
      JNB   _0a0;
      L     "DBWork".CoordSaldatura[10].Y2;
      T     "MD592";
_0a0: NOP   0;
      A     L 0.0;
      A(;
      A(;
      L     "DBWork".PP[1].NumSaldaturaAtt;
      L     10;
      ==I;
      );
      A     "AUT";
      O;
      A     "M11.2";
      A(;
      L     "DatiOP170B".PointWeldingTeachIn;
      L     11;
      ==I;
      );
      A(;
      O(;
      L     "DatiOP170B".NumeroPagina.NumeroPaginaCorrente;
      L     5;
      ==I;
      );
      O(;
      L     "DatiOP170B".NumeroPagina.NumeroPaginaCorrente;
      L     11;
      ==I;
      );
      );
      );
      =     L 0.1;
      A(;
      A     L 0.1;
      A     "DBWork".RotationTable;
      JNB   _0a1;
      L     "DBWork".CoordSaldatura[11].X1;
      T     "MD588";
      SET;
      SAVE;
      CLR;
_0a1: A     BR;
      );
      JNB   _0a2;
      L     "DBWork".CoordSaldatura[11].Y1;
      T     "MD592";
_0a2: NOP   0;
      A(;
      A     L 0.1;
      AN    "DBWork".RotationTable;
      JNB   _0a3;
      L     "DBWork".CoordSaldatura[11].X2;
      T     "MD588";
      SET;
      SAVE;
      CLR;
_0a3: A     BR;
      );
      JNB   _0a4;
      L     "DBWork".CoordSaldatura[11].Y2;
      T     "MD592";
_0a4: NOP   0;
      A     L 0.0;
      A(;
      A(;
      L     "DBWork".PP[1].NumSaldaturaAtt;
      L     11;
      ==I;
      );
      A     "AUT";
      O;
      A     "M11.2";
      A(;
      L     "DatiOP170B".PointWeldingTeachIn;
      L     12;
      ==I;
      );
      A(;
      O(;
      L     "DatiOP170B".NumeroPagina.NumeroPaginaCorrente;
      L     5;
      ==I;
      );
      O(;
      L     "DatiOP170B".NumeroPagina.NumeroPaginaCorrente;
      L     11;
      ==I;
      );
      );
      );
      =     L 0.1;
      A(;
      A     L 0.1;
      A     "DBWork".RotationTable;
      JNB   _0a5;
      L     "DBWork".CoordSaldatura[12].X1;
      T     "MD588";
      SET;
      SAVE;
      CLR;
_0a5: A     BR;
      );
      JNB   _0a6;
      L     "DBWork".CoordSaldatura[12].Y1;
      T     "MD592";
_0a6: NOP   0;
      A(;
      A     L 0.1;
      AN    "DBWork".RotationTable;
      JNB   _0a7;
      L     "DBWork".CoordSaldatura[12].X2;
      T     "MD588";
      SET;
      SAVE;
      CLR;
_0a7: A     BR;
      );
      JNB   _0a8;
      L     "DBWork".CoordSaldatura[12].Y2;
      T     "MD592";
_0a8: NOP   0;
      A     L 0.0;
      A(;
      A(;
      L     "DBWork".PP[1].NumSaldaturaAtt;
      L     12;
      ==I;
      );
      A     "AUT";
      O;
      A     "M11.2";
      A(;
      L     "DatiOP170B".PointWeldingTeachIn;
      L     13;
      ==I;
      );
      A(;
      O(;
      L     "DatiOP170B".NumeroPagina.NumeroPaginaCorrente;
      L     5;
      ==I;
      );
      O(;
      L     "DatiOP170B".NumeroPagina.NumeroPaginaCorrente;
      L     11;
      ==I;
      );
      );
      );
      =     L 0.1;
      A(;
      A     L 0.1;
      A     "DBWork".RotationTable;
      JNB   _0a9;
      L     "DBWork".CoordSaldatura[13].X1;
      T     "MD588";
      SET;
      SAVE;
      CLR;
_0a9: A     BR;
      );
      JNB   _0aa;
      L     "DBWork".CoordSaldatura[13].Y1;
      T     "MD592";
_0aa: NOP   0;
      A(;
      A     L 0.1;
      AN    "DBWork".RotationTable;
      JNB   _0ab;
      L     "DBWork".CoordSaldatura[13].X2;
      T     "MD588";
      SET;
      SAVE;
      CLR;
_0ab: A     BR;
      );
      JNB   _0ac;
      L     "DBWork".CoordSaldatura[13].Y2;
      T     "MD592";
_0ac: NOP   0;
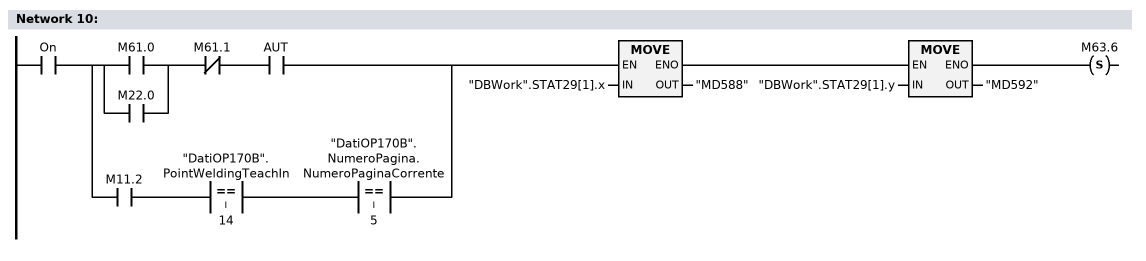
NETWORK
TITLE =
      A(;
      A     "On";
      A(;
      A(;
      O     "M61.0";
      O     "M22.0";
      );
      AN    "M61.1";
      A     "AUT";
      O;
      A     "M11.2";
      A(;
      L     "DatiOP170B".PointWeldingTeachIn;
      L     14;
      ==I;
      );
      A(;
      L     "DatiOP170B".NumeroPagina.NumeroPaginaCorrente;
      L     5;
      ==I;
      );
      );
      JNB   _0ad;
      L     "DBWork".STAT29[1].x;
      T     "MD588";
      SET;
      SAVE;
      CLR;
_0ad: A     BR;
      );
      JNB   _0ae;
      L     "DBWork".STAT29[1].y;
      T     "MD592";
      SET;
      SAVE;
      CLR;
_0ae: A     BR;
      S     "M63.6";
NETWORK
TITLE =
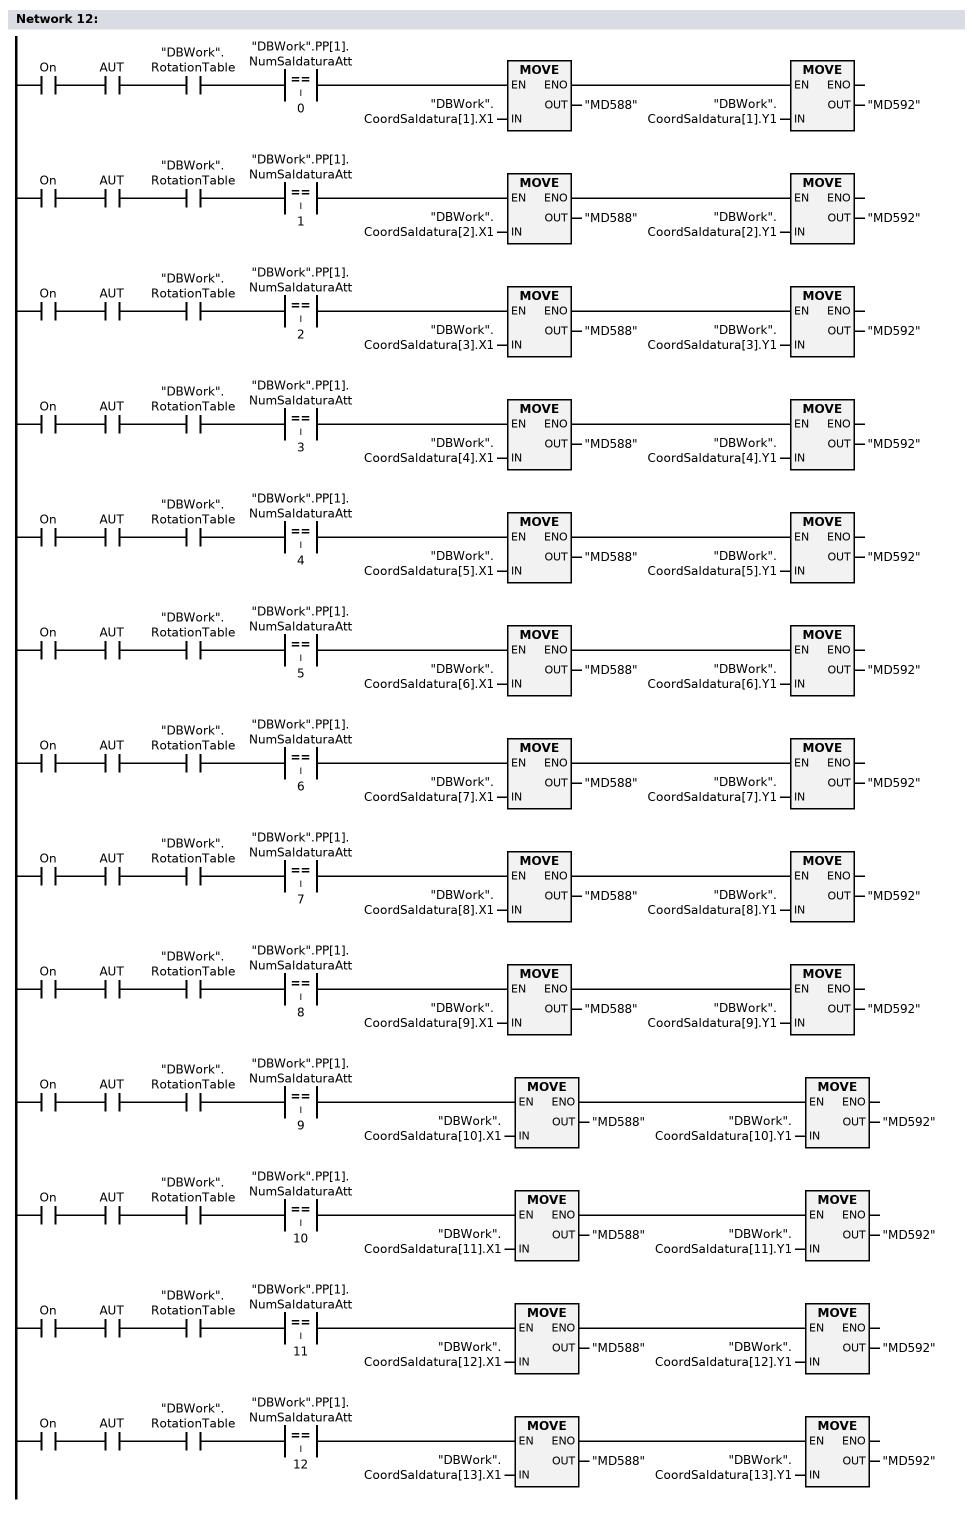
NETWORK
TITLE =
      A     "On";
      A     "AUT";
      A     "DBWork".RotationTable;
      =     L 0.0;
      A(;
      A     L 0.0;
      A(;
      L     "DBWork".PP[1].NumSaldaturaAtt;
      L     0;
      ==I;
      );
      JNB   _0af;
      L     "DBWork".CoordSaldatura[1].X1;
      T     "MD588";
      SET;
      SAVE;
      CLR;
_0af: A     BR;
      );
      JNB   _0b0;
      L     "DBWork".CoordSaldatura[1].Y1;
      T     "MD592";
_0b0: NOP   0;
      A(;
      A     L 0.0;
      A(;
      L     "DBWork".PP[1].NumSaldaturaAtt;
      L     1;
      ==I;
      );
      JNB   _0b1;
      L     "DBWork".CoordSaldatura[2].X1;
      T     "MD588";
      SET;
      SAVE;
      CLR;
_0b1: A     BR;
      );
      JNB   _0b2;
      L     "DBWork".CoordSaldatura[2].Y1;
      T     "MD592";
_0b2: NOP   0;
      A(;
      A     L 0.0;
      A(;
      L     "DBWork".PP[1].NumSaldaturaAtt;
      L     2;
      ==I;
      );
      JNB   _0b3;
      L     "DBWork".CoordSaldatura[3].X1;
      T     "MD588";
      SET;
      SAVE;
      CLR;
_0b3: A     BR;
      );
      JNB   _0b4;
      L     "DBWork".CoordSaldatura[3].Y1;
      T     "MD592";
_0b4: NOP   0;
      A(;
      A     L 0.0;
      A(;
      L     "DBWork".PP[1].NumSaldaturaAtt;
      L     3;
      ==I;
      );
      JNB   _0b5;
      L     "DBWork".CoordSaldatura[4].X1;
      T     "MD588";
      SET;
      SAVE;
      CLR;
_0b5: A     BR;
      );
      JNB   _0b6;
      L     "DBWork".CoordSaldatura[4].Y1;
      T     "MD592";
_0b6: NOP   0;
      A(;
      A     L 0.0;
      A(;
      L     "DBWork".PP[1].NumSaldaturaAtt;
      L     4;
      ==I;
      );
      JNB   _0b7;
      L     "DBWork".CoordSaldatura[5].X1;
      T     "MD588";
      SET;
      SAVE;
      CLR;
_0b7: A     BR;
      );
      JNB   _0b8;
      L     "DBWork".CoordSaldatura[5].Y1;
      T     "MD592";
_0b8: NOP   0;
      A(;
      A     L 0.0;
      A(;
      L     "DBWork".PP[1].NumSaldaturaAtt;
      L     5;
      ==I;
      );
      JNB   _0b9;
      L     "DBWork".CoordSaldatura[6].X1;
      T     "MD588";
      SET;
      SAVE;
      CLR;
_0b9: A     BR;
      );
      JNB   _0ba;
      L     "DBWork".CoordSaldatura[6].Y1;
      T     "MD592";
_0ba: NOP   0;
      A(;
      A     L 0.0;
      A(;
      L     "DBWork".PP[1].NumSaldaturaAtt;
      L     6;
      ==I;
      );
      JNB   _0bb;
      L     "DBWork".CoordSaldatura[7].X1;
      T     "MD588";
      SET;
      SAVE;
      CLR;
_0bb: A     BR;
      );
      JNB   _0bc;
      L     "DBWork".CoordSaldatura[7].Y1;
      T     "MD592";
_0bc: NOP   0;
      A(;
      A     L 0.0;
      A(;
      L     "DBWork".PP[1].NumSaldaturaAtt;
      L     7;
      ==I;
      );
      JNB   _0bd;
      L     "DBWork".CoordSaldatura[8].X1;
      T     "MD588";
      SET;
      SAVE;
      CLR;
_0bd: A     BR;
      );
      JNB   _0be;
      L     "DBWork".CoordSaldatura[8].Y1;
      T     "MD592";
_0be: NOP   0;
      A(;
      A     L 0.0;
      A(;
      L     "DBWork".PP[1].NumSaldaturaAtt;
      L     8;
      ==I;
      );
      JNB   _0bf;
      L     "DBWork".CoordSaldatura[9].X1;
      T     "MD588";
      SET;
      SAVE;
      CLR;
_0bf: A     BR;
      );
      JNB   _0c0;
      L     "DBWork".CoordSaldatura[9].Y1;
      T     "MD592";
_0c0: NOP   0;
      A(;
      A     L 0.0;
      A(;
      L     "DBWork".PP[1].NumSaldaturaAtt;
      L     9;
      ==I;
      );
      JNB   _0c1;
      L     "DBWork".CoordSaldatura[10].X1;
      T     "MD588";
      SET;
      SAVE;
      CLR;
_0c1: A     BR;
      );
      JNB   _0c2;
      L     "DBWork".CoordSaldatura[10].Y1;
      T     "MD592";
_0c2: NOP   0;
      A(;
      A     L 0.0;
      A(;
      L     "DBWork".PP[1].NumSaldaturaAtt;
      L     10;
      ==I;
      );
      JNB   _0c3;
      L     "DBWork".CoordSaldatura[11].X1;
      T     "MD588";
      SET;
      SAVE;
      CLR;
_0c3: A     BR;
      );
      JNB   _0c4;
      L     "DBWork".CoordSaldatura[11].Y1;
      T     "MD592";
_0c4: NOP   0;
      A(;
      A     L 0.0;
      A(;
      L     "DBWork".PP[1].NumSaldaturaAtt;
      L     11;
      ==I;
      );
      JNB   _0c5;
      L     "DBWork".CoordSaldatura[12].X1;
      T     "MD588";
      SET;
      SAVE;
      CLR;
_0c5: A     BR;
      );
      JNB   _0c6;
      L     "DBWork".CoordSaldatura[12].Y1;
      T     "MD592";
_0c6: NOP   0;
      A(;
      A     L 0.0;
      A(;
      L     "DBWork".PP[1].NumSaldaturaAtt;
      L     12;
      ==I;
      );
      JNB   _0c7;
      L     "DBWork".CoordSaldatura[13].X1;
      T     "MD588";
      SET;
      SAVE;
      CLR;
_0c7: A     BR;
      );
      JNB   _0c8;
      L     "DBWork".CoordSaldatura[13].Y1;
      T     "MD592";
_0c8: NOP   0;
NETWORK
TITLE =
